C05379=1020.574,11.528,-102.790,166.714,51.533,159.403
C05380=1020.580,11.777,-102.804,166.717,51.528,159.402
C05381=1020.585,12.026,-102.818,166.719,51.522,159.401
C05382=1020.591,12.276,-102.832,166.722,51.517,159.401
C05383=1020.598,12.525,-102.846,166.725,51.512,159.401
C05384=1020.603,12.775,-102.860,166.727,51.506,159.400
C05385=1020.609,13.025,-102.874,166.730,51.501,159.399
C05386=1020.615,13.274,-102.889,166.733,51.496,159.399
C05387=1020.621,13.523,-102.903,166.735,51.491,159.398
C05388=1020.627,13.773,-102.918,166.738,51.485,159.398
C05389=1020.633,14.023,-102.932,166.741,51.480,159.397
C05390=1020.638,14.272,-102.946,166.743,51.475,159.397
C05391=1020.644,14.522,-102.961,166.746,51.469,159.397
C05392=1020.649,14.771,-102.976,166.748,51.465,159.396
C05393=1020.655,15.021,-102.989,166.751,51.459,159.395
C05394=1020.661,15.270,-103.004,166.754,51.453,159.395
C05395=1020.667,15.519,-103.019,166.756,51.448,159.394
C05396=1020.673,15.769,-103.033,166.760,51.443,159.394
C05397=1020.679,16.019,-103.048,166.762,51.438,159.393
C05398=1020.684,16.269,-103.062,166.764,51.432,159.393
C05399=1020.689,16.517,-103.077,166.768,51.427,159.392
C05400=1020.696,16.768,-103.091,166.770,51.422,159.392
C05401=1020.701,17.017,-103.106,166.773,51.417,159.392
C05402=1020.708,17.266,-103.121,166.776,51.411,159.391
C05403=1020.713,17.516,-103.134,166.778,51.406,159.390
C05404=1020.719,17.765,-103.149,166.781,51.401,159.390
C05405=1020.725,18.015,-103.163,166.783,51.396,159.389
C05406=1020.730,18.264,-103.178,166.786,51.390,159.389
C05407=1020.736,18.514,-103.193,166.789,51.385,159.388
C05408=1020.742,18.764,-103.207,166.791,51.380,159.388
C05409=1020.748,19.013,-103.222,166.794,51.374,159.387
C05410=1020.754,19.262,-103.237,166.797,51.369,159.387
C05411=1020.759,19.512,-103.251,166.799,51.364,159.386
C05412=1020.765,19.762,-103.266,166.802,51.359,159.386
C05413=1020.771,20.011,-103.281,166.804,51.354,159.385
C05414=1020.776,20.260,-103.295,166.807,51.348,159.385
C05415=1020.782,20.510,-103.310,166.809,51.343,159.384
C05416=1020.788,20.759,-103.325,166.813,51.338,159.384
C05417=1020.794,21.009,-103.340,166.816,51.333,159.383
C05418=1020.799,21.259,-103.354,166.817,51.327,159.383
C05419=1020.805,21.508,-103.369,166.821,51.322,159.382
C05420=1020.811,21.757,-103.384,166.823,51.317,159.382
C05421=1020.817,22.006,-103.398,166.826,51.312,159.381
C05422=1020.823,22.256,-103.414,166.829,51.306,159.381
C05423=1020.828,22.506,-103.428,166.831,51.301,159.380
C05424=1020.834,22.756,-103.443,166.834,51.296,159.380
C05425=1020.840,23.005,-103.458,166.836,51.291,159.379
C05426=1020.846,23.255,-103.473,166.839,51.285,159.379
C05427=1020.852,23.503,-103.487,166.842,51.280,159.378
C05428=1020.857,23.754,-103.502,166.844,51.275,159.378
C05429=1020.863,24.003,-103.517,166.847,51.269,159.377
C05430=1020.869,24.253,-103.532,166.849,51.265,159.376
C05431=1020.875,24.502,-103.546,166.852,51.259,159.376
C05432=1020.881,24.752,-103.562,166.855,51.253,159.375
C05433=1020.886,25.001,-103.576,166.857,51.249,159.375
C05434=1020.893,25.250,-103.591,166.861,51.243,159.375
C05435=1020.898,25.500,-103.606,166.863,51.237,159.374
C05436=1020.904,25.750,-103.621,166.865,51.233,159.373
C05437=1020.910,25.999,-103.635,166.869,51.227,159.373
C05438=1020.915,26.249,-103.651,166.870,51.222,159.372
C05439=1020.921,26.498,-103.665,166.874,51.217,159.372
C05440=1020.928,26.782,-103.683,166.876,51.211,159.371
C05441=1020.934,27.066,-103.700,166.879,51.205,159.371
C05442=1020.941,27.350,-103.717,166.883,51.199,159.370
C05443=1020.948,27.634,-103.734,166.886,51.193,159.369
C05444=1020.953,27.883,-103.748,166.889,51.187,159.369
C05445=1020.959,28.133,-103.764,166.891,51.182,159.368
C05446=1020.965,28.382,-103.779,166.894,51.177,159.368
C05447=1020.971,28.632,-103.794,166.896,51.172,159.367
C05448=1020.976,28.881,-103.809,166.899,51.166,159.367
C05449=1020.982,29.131,-103.824,166.901,51.161,159.366
C05450=1020.988,29.380,-103.839,166.904,51.156,159.366
C05451=1020.994,29.629,-103.855,166.906,51.151,159.365
C05452=1020.999,29.879,-103.871,166.909,51.145,159.365
C05453=1021.005,30.128,-103.885,166.912,51.140,159.364
C05454=1021.011,30.378,-103.901,166.914,51.135,159.364
C05455=1021.017,30.627,-103.915,166.917,51.129,159.363
C05456=1021.022,30.877,-103.931,166.919,51.125,159.363
C05457=1021.028,31.126,-103.945,166.923,51.119,159.362
C05458=1021.034,31.376,-103.961,166.924,51.114,159.361
C05459=1021.040,31.626,-103.976,166.928,51.109,159.361
C05460=1021.045,31.875,-103.991,166.931,51.103,159.361
C05461=1021.051,32.124,-104.007,166.933,51.098,159.360
C05462=1021.057,32.373,-104.022,166.936,51.093,159.359
C05463=1021.062,32.623,-104.038,166.938,51.088,159.359
C05464=1021.069,32.873,-104.052,166.941,51.082,159.358
C05465=1021.074,33.122,-104.068,166.944,51.077,159.358
C05466=1021.080,33.372,-104.083,166.946,51.072,159.357
C05467=1021.086,33.621,-104.099,166.949,51.066,159.357
C05468=1021.092,33.870,-104.113,166.951,51.061,159.356
C05469=1021.098,34.120,-104.129,166.954,51.056,159.356
C05470=1021.103,34.370,-104.145,166.957,51.050,159.355
C05471=1021.109,34.619,-104.159,166.959,51.045,159.355
C05472=1021.115,34.868,-104.175,166.962,51.040,159.354
C05473=1021.121,35.117,-104.190,166.964,51.035,159.353
C05474=1021.126,35.367,-104.205,166.967,51.030,159.353
C05475=1021.133,35.617,-104.220,166.970,51.024,159.352
C05476=1021.138,35.866,-104.236,166.972,51.019,159.352
C05477=1021.144,36.116,-104.252,166.975,51.013,159.351
C05478=1021.150,36.365,-104.267,166.977,51.008,159.351
C05479=1021.156,36.615,-104.282,166.980,51.002,159.350
C05480=1021.162,36.864,-104.297,166.983,50.997,159.350
C05481=1021.168,37.113,-104.313,166.985,50.992,159.349
C05482=1021.173,37.363,-104.329,166.988,50.986,159.348
C05483=1021.178,37.613,-104.344,166.990,50.982,159.348
C05484=1021.184,37.862,-104.360,166.994,50.976,159.347
C05485=1021.191,38.112,-104.375,166.996,50.972,159.347
C05486=1021.196,38.360,-104.391,166.999,50.966,159.346
C05487=1021.202,38.610,-104.407,167.001,50.961,159.346
C05488=1021.207,38.860,-104.422,167.004,50.956,159.345
C05489=1021.213,39.110,-104.438,167.007,50.950,159.345
C05490=1021.218,39.359,-104.453,167.009,50.945,159.344
C05491=1021.225,39.608,-104.469,167.012,50.940,159.344
C05492=1021.231,39.858,-104.485,167.014,50.934,159.343
C05493=1021.236,40.107,-104.501,167.017,50.929,159.343
C05494=1021.242,40.357,-104.516,167.019,50.924,159.342
C05495=1021.247,40.606,-104.532,167.022,50.918,159.341
C05496=1021.254,40.856,-104.547,167.024,50.914,159.341
C05497=1021.259,41.105,-104.562,167.027,50.908,159.340
C05498=1021.265,41.354,-104.579,167.030,50.903,159.340
C05499=1021.271,41.604,-104.594,167.033,50.898,159.339
C05500=1021.276,41.853,-104.611,167.035,50.892,159.339
C05501=1021.282,42.102,-104.625,167.038,50.887,159.338
C05502=1021.288,42.352,-104.641,167.040,50.881,159.338
C05503=1021.294,42.602,-104.657,167.043,50.876,159.337
C05504=1021.300,42.885,-104.675,167.047,50.870,159.337
C05505=1021.306,43.169,-104.694,167.049,50.864,159.336
C05506=1021.313,43.453,-104.711,167.052,50.859,159.335
C05507=1021.319,43.737,-104.730,167.055,50.853,159.335
C05508=1021.325,43.987,-104.746,167.057,50.848,159.334
C05509=1021.330,44.235,-104.762,167.060,50.843,159.334
C05510=1021.336,44.485,-104.778,167.062,50.837,159.333
C05511=1021.342,44.735,-104.793,167.065,50.832,159.333
C05512=1021.347,44.984,-104.810,167.068,50.827,159.332
C05513=1021.353,45.234,-104.826,167.071,50.822,159.332
C05514=1021.358,45.483,-104.842,167.073,50.817,159.331
C05515=1021.364,45.732,-104.858,167.076,50.812,159.330
C05516=1021.370,45.982,-104.874,167.078,50.807,159.330
C05517=1021.376,46.232,-104.890,167.081,50.801,159.329
C05518=1021.382,46.481,-104.906,167.083,50.796,159.329
C05519=1021.387,46.730,-104.922,167.086,50.791,159.328
C05520=1021.393,46.979,-104.938,167.088,50.785,159.328
C05521=1021.399,47.229,-104.954,167.091,50.780,159.327
C05522=1021.404,47.479,-104.970,167.094,50.775,159.327
C05523=1021.410,47.728,-104.987,167.096,50.770,159.326
C05524=1021.415,47.977,-105.003,167.099,50.765,159.325
C05525=1021.421,48.227,-105.018,167.102,50.760,159.325
C05526=1021.427,48.476,-105.034,167.104,50.754,159.324
C05527=1021.433,48.725,-105.051,167.107,50.749,159.324
C05528=1021.439,48.975,-105.067,167.110,50.744,159.323
C05529=1021.444,49.225,-105.082,167.112,50.738,159.323
C05530=1021.450,49.473,-105.098,167.115,50.733,159.322
C05531=1021.455,49.723,-105.115,167.117,50.728,159.322
C05532=1021.461,49.972,-105.131,167.120,50.723,159.321
C05533=1021.467,50.222,-105.148,167.122,50.718,159.321
C05534=1021.472,50.472,-105.163,167.125,50.712,159.320
C05535=1021.478,50.721,-105.179,167.127,50.707,159.319
C05536=1021.484,50.970,-105.196,167.131,50.702,159.319
C05537=1021.490,51.220,-105.212,167.132,50.697,159.318
C05538=1021.496,51.468,-105.228,167.136,50.691,159.318
C05539=1021.502,51.718,-105.244,167.139,50.686,159.317
C05540=1021.506,51.968,-105.260,167.141,50.681,159.317
C05541=1021.512,52.217,-105.277,167.144,50.675,159.316
C05542=1021.518,52.467,-105.293,167.146,50.670,159.315
C05543=1021.524,52.716,-105.309,167.149,50.665,159.315
C05544=1021.530,52.965,-105.325,167.151,50.660,159.314
C05545=1021.536,53.215,-105.342,167.154,50.654,159.314
C05546=1021.542,53.464,-105.358,167.156,50.649,159.313
C05547=1021.548,53.714,-105.373,167.159,50.644,159.313
C05548=1021.553,53.964,-105.390,167.162,50.638,159.312
C05549=1021.559,54.213,-105.406,167.164,50.633,159.312
C05550=1021.564,54.462,-105.422,167.167,50.627,159.311
C05551=1021.570,54.711,-105.439,167.169,50.623,159.310
C05552=1021.576,54.960,-105.455,167.172,50.617,159.310
C05553=1021.582,55.210,-105.471,167.174,50.612,159.309
C05554=1021.588,55.459,-105.487,167.177,50.606,159.309
C05555=1021.593,55.709,-105.504,167.180,50.601,159.308
C05556=1021.599,55.958,-105.521,167.182,50.596,159.307
C05557=1021.605,56.207,-105.537,167.185,50.590,159.307
C05558=1021.611,56.457,-105.553,167.187,50.585,159.306
C05559=1021.617,56.706,-105.569,167.191,50.580,159.306
C05560=1021.623,56.955,-105.586,167.193,50.574,159.305
C05561=1021.629,57.205,-105.602,167.196,50.569,159.305
C05562=1021.635,57.454,-105.618,167.198,50.563,159.304
C05563=1021.640,57.704,-105.635,167.200,50.558,159.303
C05564=1021.646,57.953,-105.651,167.204,50.553,159.303
C05565=1021.652,58.202,-105.667,167.206,50.547,159.302
C05566=1021.658,58.452,-105.684,167.209,50.542,159.302
C05567=1021.664,58.701,-105.700,167.212,50.536,159.301
C05568=1021.671,58.985,-105.719,167.214,50.531,159.300
C05569=1021.677,59.270,-105.737,167.217,50.525,159.300
C05570=1021.684,59.552,-105.756,167.221,50.518,159.299
C05571=1021.691,59.836,-105.774,167.224,50.512,159.299
C05572=1021.696,60.086,-105.790,167.225,50.507,159.298
C05573=1021.702,60.335,-105.807,167.229,50.502,159.297
C05574=1021.708,60.584,-105.823,167.232,50.496,159.297
C05575=1021.714,60.834,-105.840,167.233,50.490,159.296
C05576=1021.720,61.083,-105.856,167.237,50.485,159.296
C05577=1021.725,61.333,-105.872,167.240,50.479,159.295
C05578=1021.732,61.583,-105.889,167.241,50.474,159.294
C05579=1021.738,61.831,-105.906,167.245,50.469,159.294
C05580=1021.744,62.081,-105.922,167.248,50.463,159.293
C05581=1021.749,62.330,-105.939,167.250,50.458,159.293
C05582=1021.755,62.580,-105.955,167.253,50.453,159.292
C05583=1021.761,62.829,-105.972,167.254,50.447,159.291
C05584=1021.767,63.078,-105.988,167.258,50.442,159.291
C05585=1021.773,63.328,-106.005,167.261,50.436,159.290
C05586=1021.779,63.577,-106.022,167.263,50.431,159.290
C05587=1021.785,63.826,-106.038,167.266,50.426,159.289
C05588=1021.793,64.185,-106.062,167.269,50.418,159.288
C05589=1021.801,64.542,-106.087,167.273,50.410,159.287
C05590=1021.809,64.899,-106.110,167.277,50.403,159.287
C05591=1021.817,65.257,-106.134,167.281,50.396,159.286
C05592=1021.823,65.506,-106.151,167.283,50.390,159.285
C05593=1021.829,65.755,-106.168,167.286,50.385,159.285
C05594=1021.835,66.005,-106.184,167.289,50.379,159.284
C05595=1021.841,66.254,-106.202,167.291,50.375,159.283
C05596=1021.847,66.504,-106.218,167.294,50.369,159.283
C05597=1021.852,66.753,-106.235,167.296,50.364,159.282
C05598=1021.858,67.002,-106.252,167.299,50.358,159.282
C05599=1021.863,67.252,-106.269,167.301,50.353,159.281
C05600=1021.869,67.501,-106.285,167.304,50.348,159.280
C05601=1021.875,67.750,-106.303,167.307,50.343,159.280
C05602=1021.881,68.000,-106.319,167.309,50.337,159.279
C05603=1021.886,68.249,-106.337,167.312,50.331,159.279
C05604=1021.893,68.499,-106.353,167.314,50.327,159.278
C05605=1021.898,68.748,-106.370,167.318,50.322,159.278
C05606=1021.904,68.997,-106.387,167.320,50.316,159.277
C05607=1021.909,69.247,-106.404,167.323,50.311,159.276
C05608=1021.915,69.496,-106.421,167.325,50.306,159.276
C05609=1021.921,69.745,-106.438,167.328,50.300,159.275
C05610=1021.927,69.995,-106.456,167.330,50.295,159.275
C05611=1021.932,70.244,-106.473,167.333,50.290,159.274
C05612=1021.939,70.493,-106.489,167.336,50.284,159.274
C05613=1021.944,70.743,-106.506,167.338,50.279,159.273
C05614=1021.949,70.992,-106.524,167.341,50.274,159.272
C05615=1021.955,71.241,-106.540,167.343,50.269,159.272
C05616=1021.961,71.491,-106.558,167.346,50.263,159.271
C05617=1021.967,71.741,-106.575,167.349,50.258,159.271
C05618=1021.973,71.989,-106.592,167.351,50.253,159.270
C05619=1021.978,72.238,-106.609,167.354,50.248,159.269
C05620=1021.984,72.488,-106.626,167.357,50.242,159.269
C05621=1021.989,72.737,-106.644,167.359,50.237,159.268
C05622=1021.996,72.987,-106.661,167.362,50.232,159.268
C05623=1022.001,73.236,-106.678,167.365,50.227,159.267
C05624=1022.006,73.486,-106.695,167.367,50.221,159.266
C05625=1022.013,73.735,-106.712,167.370,50.216,159.266
C05626=1022.019,73.984,-106.730,167.372,50.211,159.265
C05627=1022.024,74.234,-106.747,167.375,50.205,159.265
C05628=1022.029,74.446,-106.761,167.378,50.201,159.264
C05629=1022.034,74.658,-106.776,167.380,50.196,159.264
C05630=1022.039,74.871,-106.790,167.382,50.191,159.263
C05631=1022.044,75.083,-106.805,167.384,50.188,159.263
C05632=1022.049,75.295,-106.820,167.386,50.183,159.262
C05633=1022.054,75.508,-106.835,167.388,50.178,159.262
C05634=1022.058,75.720,-106.849,167.390,50.173,159.261
C05635=1022.063,75.933,-106.864,167.393,50.169,159.261
C05636=1022.069,76.182,-106.882,167.396,50.163,159.260
C05637=1022.075,76.431,-106.898,167.398,50.159,159.260
C05638=1022.081,76.681,-106.916,167.401,50.153,159.259
C05639=1022.087,76.930,-106.933,167.403,50.148,159.258
C05640=1022.092,77.179,-106.951,167.406,50.142,159.258
C05641=1022.097,77.429,-106.968,167.409,50.138,159.257
C05642=1022.103,77.679,-106.986,167.411,50.132,159.257
C05643=1022.109,77.928,-107.003,167.414,50.127,159.256
C05644=1022.114,78.177,-107.021,167.417,50.122,159.255
C05645=1022.120,78.426,-107.038,167.420,50.116,159.255
C05646=1022.126,78.676,-107.056,167.422,50.111,159.254
C05647=1022.131,78.925,-107.073,167.425,50.106,159.254
C05648=1022.137,79.174,-107.091,167.427,50.101,159.253
C05649=1022.143,79.424,-107.109,167.430,50.096,159.253
C05650=1022.149,79.673,-107.126,167.433,50.091,159.252
C05651=1022.155,79.922,-107.143,167.435,50.085,159.252
C05652=1022.160,80.171,-107.160,167.438,50.080,159.251
C05653=1022.166,80.421,-107.178,167.441,50.075,159.250
C05654=1022.172,80.670,-107.196,167.443,50.070,159.250
C05655=1022.177,80.919,-107.213,167.446,50.064,159.249
C05656=1022.183,81.169,-107.231,167.448,50.059,159.249
C05657=1022.189,81.418,-107.249,167.451,50.054,159.248
C05658=1022.194,81.667,-107.266,167.453,50.049,159.247
C05659=1022.200,81.916,-107.284,167.456,50.043,159.247
C05660=1022.206,82.166,-107.302,167.459,50.038,159.246
C05661=1022.211,82.415,-107.319,167.461,50.033,159.246
C05662=1022.217,82.664,-107.337,167.465,50.028,159.245
C05663=1022.223,82.914,-107.354,167.467,50.022,159.244
C05664=1022.228,83.163,-107.372,167.470,50.017,159.244
C05665=1022.234,83.412,-107.389,167.472,50.012,159.243
C05666=1022.240,83.662,-107.407,167.475,50.007,159.243
C05667=1022.245,83.911,-107.425,167.478,50.001,159.242
C05668=1022.252,84.161,-107.443,167.480,49.996,159.241
C05669=1022.257,84.410,-107.460,167.483,49.991,159.241
C05670=1022.263,84.659,-107.478,167.485,49.985,159.240
C05671=1022.269,84.909,-107.496,167.488,49.980,159.240
C05672=1022.274,85.158,-107.513,167.490,49.975,159.239
C05673=1022.280,85.407,-107.531,167.494,49.970,159.239
C05674=1022.286,85.656,-107.549,167.497,49.964,159.238
C05675=1022.291,85.906,-107.566,167.499,49.959,159.237
C05676=1022.297,86.155,-107.584,167.502,49.953,159.237
C05677=1022.303,86.404,-107.602,167.504,49.948,159.236
C05678=1022.309,86.653,-107.619,167.507,49.943,159.236
C05679=1022.315,86.903,-107.637,167.510,49.937,159.235
C05680=1022.320,87.152,-107.655,167.512,49.933,159.234
C05681=1022.326,87.402,-107.673,167.515,49.927,159.234
C05682=1022.332,87.651,-107.690,167.517,49.921,159.233
C05683=1022.338,87.899,-107.709,167.520,49.916,159.233
C05684=1022.344,88.149,-107.727,167.523,49.911,159.232
C05685=1022.349,88.398,-107.744,167.526,49.906,159.231
C05686=1022.355,88.648,-107.762,167.529,49.900,159.231
C05687=1022.361,88.897,-107.780,167.530,49.895,159.230
C05688=1022.367,89.147,-107.798,167.534,49.890,159.230
C05689=1022.372,89.396,-107.816,167.537,49.884,159.229
C05690=1022.378,89.646,-107.834,167.539,49.879,159.228
C05691=1022.383,89.895,-107.851,167.542,49.874,159.228
C05692=1022.389,90.143,-107.870,167.544,49.869,159.227
C05693=1022.395,90.393,-107.888,167.547,49.863,159.227
C05694=1022.400,90.642,-107.906,167.549,49.859,159.226
C05695=1022.406,90.892,-107.924,167.552,49.853,159.225
C05696=1022.413,91.175,-107.944,167.555,49.847,159.225
C05697=1022.419,91.459,-107.965,167.558,49.841,159.224
C05698=1022.425,91.742,-107.986,167.561,49.836,159.224
C05699=1022.432,92.026,-108.007,167.565,49.829,159.223
C05700=1022.437,92.275,-108.025,167.567,49.824,159.222
C05701=1022.443,92.525,-108.043,167.570,49.819,159.222
C05702=1022.448,92.774,-108.061,167.572,49.814,159.221
C05703=1022.455,93.023,-108.079,167.575,49.808,159.221
C05704=1022.460,93.272,-108.097,167.578,49.804,159.220
C05705=1022.466,93.522,-108.115,167.581,49.798,159.219
C05706=1022.471,93.771,-108.134,167.584,49.793,159.219
C05707=1022.477,94.020,-108.151,167.586,49.787,159.218
C05708=1022.483,94.270,-108.169,167.589,49.782,159.218
C05709=1022.488,94.518,-108.188,167.591,49.777,159.217
C05710=1022.494,94.768,-108.206,167.594,49.772,159.217
C05711=1022.500,95.016,-108.224,167.596,49.767,159.216
C05712=1022.505,95.267,-108.243,167.600,49.762,159.215
C05713=1022.511,95.516,-108.261,167.603,49.756,159.215
C05714=1022.517,95.765,-108.279,167.605,49.751,159.214
C05715=1022.523,96.015,-108.298,167.608,49.746,159.214
C05716=1022.528,96.264,-108.315,167.610,49.740,159.213
C05717=1022.535,96.513,-108.334,167.613,49.735,159.212
C05718=1022.539,96.762,-108.352,167.616,49.729,159.212
C05719=1022.546,97.011,-108.371,167.618,49.725,159.211
C05720=1022.551,97.260,-108.388,167.621,49.719,159.211
C05721=1022.557,97.510,-108.408,167.624,49.714,159.210
C05722=1022.563,97.759,-108.425,167.627,49.709,159.209
C05723=1022.569,98.009,-108.443,167.630,49.703,159.209
C05724=1022.574,98.258,-108.462,167.632,49.698,159.208
C05725=1022.580,98.507,-108.480,167.635,49.693,159.207
C05726=1022.586,98.756,-108.498,167.638,49.688,159.207
C05727=1022.591,99.006,-108.517,167.640,49.682,159.206
C05728=1022.597,99.255,-108.535,167.643,49.677,159.206
C05729=1022.603,99.504,-108.553,167.645,49.672,159.205
C05730=1022.609,99.753,-108.572,167.648,49.666,159.204
C05731=1022.614,100.003,-108.591,167.652,49.661,159.204
C05732=1022.620,100.252,-108.609,167.654,49.657,159.203
C05733=1022.626,100.501,-108.628,167.657,49.651,159.203
C05734=1022.631,100.750,-108.646,167.659,49.646,159.202
C05735=1022.637,101.000,-108.665,167.662,49.640,159.202
C05736=1022.642,101.249,-108.683,167.665,49.636,159.201
C05737=1022.648,101.498,-108.702,167.668,49.630,159.200
C05738=1022.654,101.747,-108.721,167.670,49.625,159.200
C05739=1022.659,101.997,-108.739,167.673,49.620,159.199
C05740=1022.665,102.246,-108.758,167.676,49.615,159.199
C05741=1022.670,102.495,-108.777,167.678,49.609,159.198
C05742=1022.676,102.744,-108.795,167.681,49.604,159.198
C05743=1022.682,102.994,-108.814,167.683,49.599,159.197
C05744=1022.687,103.243,-108.833,167.687,49.594,159.196
C05745=1022.693,103.492,-108.851,167.690,49.588,159.196
C05746=1022.699,103.742,-108.870,167.692,49.584,159.195
C05747=1022.704,103.990,-108.888,167.695,49.578,159.195
C05748=1022.710,104.240,-108.907,167.697,49.573,159.194
C05749=1022.715,104.489,-108.926,167.700,49.568,159.193
C05750=1022.721,104.738,-108.944,167.703,49.563,159.193
C05751=1022.727,104.988,-108.964,167.706,49.557,159.192
C05752=1022.732,105.237,-108.982,167.709,49.552,159.192
C05753=1022.738,105.486,-109.000,167.711,49.547,159.191
C05754=1022.744,105.735,-109.020,167.714,49.542,159.191
C05755=1022.750,105.984,-109.038,167.717,49.536,159.190
C05756=1022.755,106.233,-109.057,167.720,49.532,159.189
C05757=1022.761,106.483,-109.076,167.723,49.526,159.189
C05758=1022.767,106.732,-109.094,167.725,49.521,159.188
C05759=1022.772,106.981,-109.113,167.728,49.516,159.188
C05760=1022.779,107.265,-109.134,167.731,49.510,159.187
C05761=1022.785,107.549,-109.155,167.735,49.504,159.186
C05762=1022.792,107.832,-109.177,167.737,49.498,159.186
C05763=1022.799,108.116,-109.199,167.740,49.492,159.185
C05764=1022.804,108.365,-109.217,167.743,49.486,159.184
C05765=1022.810,108.614,-109.236,167.746,49.482,159.184
C05766=1022.815,108.864,-109.255,167.749,49.476,159.183
C05767=1022.821,109.113,-109.273,167.752,49.471,159.183
C05768=1022.827,109.362,-109.292,167.754,49.466,159.182
C05769=1022.833,109.612,-109.312,167.757,49.460,159.181
C05770=1022.839,109.861,-109.330,167.760,49.455,159.181
C05771=1022.844,110.109,-109.349,167.762,49.450,159.180
C05772=1022.850,110.359,-109.368,167.766,49.445,159.180
C05773=1022.856,110.608,-109.388,167.769,49.439,159.179
C05774=1022.861,110.858,-109.407,167.771,49.434,159.178
C05775=1022.867,111.106,-109.425,167.774,49.429,159.178
C05776=1022.873,111.356,-109.444,167.776,49.424,159.177
C05777=1022.878,111.605,-109.464,167.779,49.419,159.177
C05778=1022.884,111.854,-109.483,167.783,49.414,159.176
C05779=1022.889,112.103,-109.502,167.785,49.408,159.175
C05780=1022.895,112.353,-109.521,167.788,49.403,159.175
C05781=1022.901,112.602,-109.540,167.791,49.398,159.174
C05782=1022.906,112.851,-109.559,167.793,49.393,159.174
C05783=1022.911,113.100,-109.578,167.797,49.388,159.173
C05784=1022.917,113.350,-109.598,167.799,49.383,159.173
C05785=1022.923,113.599,-109.617,167.802,49.378,159.172
C05786=1022.928,113.848,-109.636,167.804,49.373,159.172
C05787=1022.933,114.097,-109.655,167.807,49.367,159.171
C05788=1022.939,114.346,-109.675,167.810,49.363,159.170
C05789=1022.945,114.595,-109.694,167.813,49.358,159.170
C05790=1022.951,114.845,-109.713,167.816,49.352,159.169
C05791=1022.956,115.094,-109.732,167.818,49.348,159.169
C05792=1022.961,115.343,-109.752,167.822,49.342,159.168
C05793=1022.967,115.593,-109.771,167.824,49.337,159.168
C05794=1022.973,115.842,-109.791,167.827,49.332,159.167
C05795=1022.978,116.091,-109.811,167.830,49.327,159.166
C05796=1022.983,116.340,-109.829,167.833,49.322,159.166
C05797=1022.989,116.589,-109.849,167.836,49.317,159.165
C05798=1022.995,116.838,-109.869,167.838,49.312,159.165
C05799=1023.001,117.087,-109.888,167.841,49.307,159.164
C05800=1023.006,117.337,-109.907,167.844,49.301,159.164
C05801=1023.011,117.586,-109.927,167.847,49.297,159.163
C05802=1023.017,117.835,-109.947,167.850,49.292,159.163
C05803=1023.022,118.084,-109.966,167.852,49.286,159.162
C05804=1023.028,118.334,-109.985,167.855,49.281,159.161
C05805=1023.034,118.583,-110.004,167.858,49.276,159.161
C05806=1023.039,118.831,-110.024,167.861,49.271,159.160
C05807=1023.045,119.081,-110.043,167.864,49.265,159.160
C05808=1023.051,119.330,-110.062,167.867,49.260,159.159
C05809=1023.056,119.579,-110.082,167.869,49.256,159.159
C05810=1023.062,119.829,-110.102,167.872,49.250,159.158
C05811=1023.067,120.078,-110.121,167.876,49.245,159.157
C05812=1023.073,120.327,-110.141,167.878,49.240,159.157
C05813=1023.078,120.576,-110.160,167.881,49.235,159.156
C05814=1023.084,120.825,-110.179,167.883,49.230,159.156
C05815=1023.090,121.074,-110.199,167.887,49.225,159.155
C05816=1023.096,121.323,-110.219,167.890,49.219,159.154
C05817=1023.101,121.573,-110.238,167.892,49.215,159.154
C05818=1023.107,121.822,-110.258,167.895,49.210,159.153
C05819=1023.112,122.071,-110.278,167.898,49.204,159.153
C05820=1023.118,122.321,-110.297,167.901,49.199,159.152
C05821=1023.124,122.569,-110.317,167.904,49.194,159.152
C05822=1023.130,122.819,-110.336,167.907,49.189,159.151
C05823=1023.135,123.068,-110.355,167.910,49.183,159.150
C05824=1023.141,123.351,-110.377,167.913,49.178,159.150
C05825=1023.148,123.635,-110.400,167.916,49.172,159.149
C05826=1023.154,123.919,-110.422,167.920,49.165,159.148
C05827=1023.161,124.202,-110.444,167.923,49.160,159.148
C05828=1023.167,124.451,-110.464,167.926,49.155,159.147
C05829=1023.172,124.701,-110.484,167.928,49.150,159.147
C05830=1023.178,124.950,-110.504,167.932,49.145,159.146
C05831=1023.184,125.199,-110.523,167.935,49.139,159.146
C05832=1023.190,125.448,-110.543,167.937,49.134,159.145
C05833=1023.195,125.697,-110.563,167.940,49.129,159.144
C05834=1023.201,125.946,-110.582,167.943,49.124,159.144
C05835=1023.207,126.196,-110.602,167.947,49.118,159.143
C05836=1023.212,126.445,-110.622,167.949,49.114,159.143
C05837=1023.218,126.694,-110.642,167.952,49.108,159.142
C05838=1023.224,126.943,-110.661,167.955,49.103,159.142
C05839=1023.230,127.192,-110.681,167.957,49.098,159.141
C05840=1023.236,127.441,-110.701,167.961,49.093,159.140
C05841=1023.241,127.691,-110.720,167.964,49.087,159.140
C05842=1023.247,127.939,-110.740,167.967,49.082,159.139
C05843=1023.252,128.189,-110.760,167.969,49.077,159.139
C05844=1023.258,128.438,-110.780,167.973,49.072,159.138
C05845=1023.264,128.687,-110.799,167.976,49.067,159.137
C05846=1023.270,128.936,-110.819,167.979,49.061,159.137
C05847=1023.276,129.186,-110.838,167.981,49.056,159.136
C05848=1023.282,129.434,-110.858,167.984,49.051,159.136
C05849=1023.288,129.683,-110.878,167.987,49.046,159.135
C05850=1023.292,129.933,-110.898,167.990,49.040,159.134
C05851=1023.298,130.182,-110.918,167.993,49.036,159.134
C05852=1023.304,130.431,-110.938,167.996,49.031,159.133
C05853=1023.309,130.680,-110.958,167.999,49.025,159.133
C05854=1023.315,130.929,-110.978,168.003,49.020,159.132
C05855=1023.321,131.178,-110.998,168.005,49.015,159.132
C05856=1023.327,131.427,-111.018,168.008,49.010,159.131
C05857=1023.332,131.677,-111.038,168.011,49.005,159.131
C05858=1023.338,131.926,-111.058,168.013,49.000,159.130
C05859=1023.343,132.175,-111.078,168.017,48.995,159.129
C05860=1023.349,132.424,-111.098,168.020,48.990,159.129
C05861=1023.354,132.673,-111.119,168.022,48.985,159.128
C05862=1023.360,132.922,-111.138,168.026,48.980,159.128
C05863=1023.365,133.171,-111.159,168.029,48.974,159.127
C05864=1023.372,133.421,-111.179,168.032,48.969,159.127
C05865=1023.377,133.670,-111.200,168.034,48.965,159.126
C05866=1023.383,133.919,-111.220,168.038,48.959,159.125
C05867=1023.388,134.168,-111.240,168.041,48.954,159.125
C05868=1023.394,134.417,-111.259,168.043,48.950,159.124
C05869=1023.399,134.666,-111.280,168.046,48.944,159.124
C05870=1023.405,134.915,-111.300,168.050,48.939,159.123
C05871=1023.410,135.164,-111.320,168.053,48.934,159.123
C05872=1023.416,135.413,-111.340,168.055,48.929,159.122
C05873=1023.422,135.662,-111.361,168.059,48.924,159.122
C05874=1023.428,135.911,-111.381,168.062,48.919,159.121
C05875=1023.433,136.161,-111.402,168.065,48.914,159.121
C05876=1023.439,136.410,-111.421,168.067,48.908,159.120
C05877=1023.444,136.659,-111.442,168.071,48.903,159.119
C05878=1023.450,136.908,-111.462,168.074,48.899,159.119
C05879=1023.456,137.157,-111.482,168.077,48.893,159.118
C05880=1023.461,137.407,-111.503,168.079,48.888,159.118
C05881=1023.467,137.655,-111.523,168.083,48.884,159.117
C05882=1023.473,137.905,-111.544,168.086,48.878,159.117
C05883=1023.479,138.154,-111.564,168.089,48.873,159.116
C05884=1023.484,138.403,-111.584,168.092,48.868,159.116
C05885=1023.489,138.652,-111.605,168.095,48.863,159.115
C05886=1023.495,138.901,-111.625,168.098,48.858,159.114
C05887=1023.500,139.150,-111.645,168.101,48.853,159.114
C05888=1023.507,139.434,-111.669,168.105,48.848,159.113
C05889=1023.513,139.718,-111.693,168.108,48.842,159.113
C05890=1023.520,140.001,-111.716,168.112,48.836,159.112
C05891=1023.526,140.284,-111.739,168.115,48.831,159.111
C05892=1023.532,140.533,-111.760,168.118,48.825,159.111
C05893=1023.537,140.782,-111.781,168.121,48.820,159.110
C05894=1023.543,141.031,-111.801,168.124,48.816,159.110
C05895=1023.549,141.281,-111.821,168.127,48.810,159.109
C05896=1023.554,141.530,-111.842,168.130,48.805,159.109
C05897=1023.559,141.779,-111.863,168.134,48.800,159.108
C05898=1023.565,142.027,-111.883,168.136,48.796,159.108
C05899=1023.571,142.276,-111.904,168.139,48.790,159.107
C05900=1023.577,142.526,-111.925,168.142,48.785,159.107
C05901=1023.582,142.775,-111.945,168.146,48.780,159.106
C05902=1023.588,143.024,-111.965,168.148,48.775,159.105
C05903=1023.593,143.273,-111.987,168.151,48.770,159.105
C05904=1023.599,143.522,-112.007,168.155,48.765,159.104
C05905=1023.605,143.772,-112.028,168.158,48.760,159.104
C05906=1023.611,144.020,-112.048,168.161,48.755,159.103
C05907=1023.616,144.269,-112.069,168.164,48.750,159.103
C05908=1023.622,144.519,-112.090,168.167,48.745,159.102
C05909=1023.627,144.768,-112.111,168.170,48.740,159.102
C05910=1023.632,145.017,-112.131,168.174,48.735,159.101
C05911=1023.639,145.265,-112.152,168.177,48.730,159.100
C05912=1023.645,145.515,-112.173,168.179,48.725,159.100
C05913=1023.650,145.764,-112.193,168.182,48.720,159.099
C05914=1023.655,146.013,-112.214,168.185,48.715,159.099
C05915=1023.661,146.262,-112.236,168.189,48.710,159.098
C05916=1023.667,146.512,-112.256,168.192,48.705,159.098
C05917=1023.672,146.760,-112.277,168.195,48.700,159.097
C05918=1023.678,147.009,-112.297,168.198,48.695,159.097
C05919=1023.684,147.259,-112.318,168.201,48.690,159.096
C05920=1023.689,147.507,-112.340,168.205,48.685,159.096
C05921=1023.695,147.756,-112.360,168.208,48.680,159.095
C05922=1023.701,148.006,-112.382,168.210,48.676,159.095
C05923=1023.706,148.255,-112.402,168.214,48.670,159.094
C05924=1023.712,148.503,-112.424,168.217,48.665,159.094
C05925=1023.717,148.752,-112.444,168.220,48.660,159.093
C05926=1023.723,149.002,-112.465,168.224,48.655,159.093
C05927=1023.728,149.251,-112.486,168.226,48.650,159.092
C05928=1023.734,149.500,-112.507,168.229,48.645,159.091
C05929=1023.740,149.749,-112.528,168.233,48.641,159.091
C05930=1023.745,149.998,-112.549,168.236,48.636,159.090
C05931=1023.751,150.247,-112.570,168.240,48.631,159.090
C05932=1023.756,150.496,-112.593,168.242,48.626,159.089
C05933=1023.761,150.745,-112.613,168.245,48.621,159.089
C05934=1023.767,150.994,-112.634,168.249,48.616,159.088
C05935=1023.773,151.244,-112.655,168.252,48.611,159.088
C05936=1023.778,151.492,-112.677,168.255,48.606,159.087
C05937=1023.784,151.742,-112.697,168.258,48.601,159.087
C05938=1023.790,151.990,-112.719,168.261,48.596,159.086
C05939=1023.795,152.240,-112.739,168.264,48.591,159.086
C05940=1023.801,152.489,-112.761,168.268,48.586,159.085
C05941=1023.807,152.737,-112.782,168.271,48.581,159.085
C05942=1023.812,152.986,-112.803,168.274,48.576,159.084
C05943=1023.818,153.236,-112.824,168.278,48.571,159.084
C05944=1023.824,153.484,-112.846,168.280,48.567,159.083
C05945=1023.830,153.734,-112.867,168.284,48.562,159.083
C05946=1023.834,153.983,-112.888,168.287,48.557,159.082
C05947=1023.841,154.232,-112.910,168.290,48.551,159.081
C05948=1023.846,154.481,-112.931,168.294,48.547,159.081
C05949=1023.851,154.730,-112.952,168.297,48.542,159.080
C05950=1023.858,154.979,-112.974,168.299,48.537,159.080
C05951=1023.862,155.228,-112.995,168.303,48.532,159.079
C05952=1023.869,155.512,-113.019,168.307,48.527,159.079
C05953=1023.875,155.794,-113.044,168.310,48.521,159.078
C05954=1023.882,156.078,-113.067,168.314,48.515,159.078
C05955=1023.888,156.360,-113.092,168.317,48.510,159.077
C05956=1023.894,156.610,-113.113,168.321,48.505,159.077
C05957=1023.899,156.858,-113.135,168.324,48.500,159.076
C05958=1023.905,157.108,-113.156,168.328,48.495,159.076
C05959=1023.910,157.357,-113.177,168.331,48.490,159.075
C05960=1023.917,157.606,-113.199,168.334,48.486,159.075
C05961=1023.921,157.855,-113.221,168.338,48.480,159.074
C05962=1023.928,158.104,-113.243,168.341,48.475,159.074
C05963=1023.933,158.352,-113.264,168.343,48.471,159.073
C05964=1023.939,158.602,-113.285,168.347,48.466,159.072
C05965=1023.945,158.851,-113.306,168.350,48.461,159.072
C05966=1023.950,159.100,-113.328,168.354,48.456,159.072
C05967=1023.956,159.349,-113.350,168.357,48.451,159.071
C05968=1023.961,159.598,-113.372,168.361,48.447,159.071
C05969=1023.967,159.847,-113.393,168.364,48.442,159.070
C05970=1023.972,160.096,-113.415,168.367,48.437,159.070
C05971=1023.977,160.345,-113.437,168.370,48.432,159.069
C05972=1023.983,160.594,-113.459,168.373,48.428,159.069
C05973=1023.988,160.843,-113.481,168.377,48.423,159.068
C05974=1023.993,161.091,-113.503,168.380,48.418,159.068
C05975=1023.999,161.341,-113.525,168.383,48.413,159.067
C05976=1024.004,161.589,-113.547,168.386,48.409,159.067
C05977=1024.009,161.839,-113.569,168.390,48.404,159.066
C05978=1024.015,162.087,-113.590,168.393,48.400,159.066
C05979=1024.020,162.337,-113.612,168.397,48.395,159.065
C05980=1024.025,162.585,-113.635,168.400,48.390,159.065
C05981=1024.032,162.834,-113.657,168.403,48.385,159.064
C05982=1024.037,163.084,-113.679,168.406,48.381,159.064
C05983=1024.042,163.333,-113.701,168.410,48.376,159.063
C05984=1024.048,163.582,-113.722,168.413,48.371,159.063
C05985=1024.053,163.831,-113.744,168.417,48.366,159.062
C05986=1024.059,164.080,-113.767,168.420,48.361,159.062
C05987=1024.064,164.328,-113.788,168.423,48.357,159.061
C05988=1024.070,164.578,-113.811,168.426,48.352,159.061
C05989=1024.074,164.826,-113.833,168.429,48.347,159.060
C05990=1024.081,165.075,-113.855,168.433,48.342,159.060
C05991=1024.086,165.325,-113.877,168.436,48.338,159.059
C05992=1024.091,165.573,-113.899,168.440,48.333,159.059
C05993=1024.097,165.823,-113.921,168.443,48.329,159.059
C05994=1024.102,166.071,-113.943,168.447,48.324,159.058
C05995=1024.108,166.320,-113.965,168.450,48.319,159.058
C05996=1024.113,166.569,-113.987,168.454,48.314,159.057
C05997=1024.119,166.818,-114.010,168.457,48.309,159.057
C05998=1024.125,167.067,-114.032,168.460,48.305,159.056
C05999=1024.130,167.316,-114.053,168.463,48.300,159.056
C06000=1024.135,167.565,-114.075,168.467,48.295,159.055
C06001=1024.141,167.814,-114.098,168.470,48.290,159.055
C06002=1024.146,168.063,-114.120,168.474,48.286,159.054
C06003=1024.153,168.311,-114.143,168.477,48.281,159.054
C06004=1024.158,168.561,-114.165,168.480,48.276,159.053
C06005=1024.163,168.810,-114.187,168.484,48.271,159.053
C06006=1024.169,169.058,-114.209,168.488,48.267,159.052
C06007=1024.175,169.308,-114.231,168.491,48.262,159.052
C06008=1024.179,169.557,-114.253,168.495,48.258,159.052
C06009=1024.186,169.805,-114.275,168.498,48.253,159.051
C06010=1024.191,170.055,-114.298,168.502,48.248,159.051
C06011=1024.197,170.303,-114.320,168.505,48.243,159.050
C06012=1024.203,170.552,-114.342,168.509,48.238,159.050
C06013=1024.208,170.802,-114.364,168.512,48.234,159.049
C06014=1024.213,171.050,-114.387,168.515,48.229,159.049
C06015=1024.219,171.299,-114.409,168.519,48.224,159.048
C06016=1024.226,171.582,-114.434,168.522,48.219,159.048
C06017=1024.232,171.865,-114.460,168.527,48.213,159.047
C06018=1024.238,172.147,-114.484,168.531,48.208,159.047
C06019=1024.245,172.431,-114.510,168.534,48.203,159.046
C06020=1024.250,172.680,-114.533,168.538,48.198,159.046
C06021=1024.256,172.928,-114.555,168.541,48.193,159.045
C06022=1024.262,173.177,-114.577,168.545,48.189,159.045
C06023=1024.267,173.426,-114.600,168.548,48.184,159.044
C06024=1024.273,173.676,-114.622,168.551,48.179,159.044
C06025=1024.279,173.924,-114.644,168.555,48.174,159.043
C06026=1024.284,174.173,-114.667,168.558,48.169,159.043
C06027=1024.290,174.422,-114.689,168.563,48.164,159.042
C06028=1024.296,174.671,-114.712,168.566,48.160,159.042
C06029=1024.302,174.920,-114.734,168.570,48.155,159.041
C06030=1024.308,175.169,-114.757,168.574,48.151,159.041
C06031=1024.312,175.418,-114.779,168.577,48.146,159.040
C06032=1024.319,175.667,-114.801,168.581,48.141,159.040
C06033=1024.325,175.915,-114.824,168.584,48.136,159.040
C06034=1024.330,176.165,-114.846,168.588,48.132,159.039
C06035=1024.336,176.414,-114.868,168.591,48.127,159.039
C06036=1024.342,176.662,-114.891,168.594,48.122,159.038
C06037=1024.347,176.911,-114.913,168.598,48.117,159.038
C06038=1024.353,177.160,-114.936,168.601,48.112,159.037
C06039=1024.359,177.409,-114.959,168.605,48.108,159.037
C06040=1024.365,177.658,-114.981,168.608,48.103,159.036
C06041=1024.370,177.907,-115.004,168.613,48.098,159.036
C06042=1024.377,178.156,-115.026,168.617,48.094,159.035
C06043=1024.382,178.405,-115.048,168.620,48.089,159.035
C06044=1024.388,178.654,-115.071,168.624,48.084,159.034
C06045=1024.393,178.902,-115.094,168.627,48.079,159.034
C06046=1024.400,179.151,-115.116,168.631,48.075,159.033
C06047=1024.405,179.400,-115.138,168.634,48.070,159.033
C06048=1024.411,179.649,-115.161,168.638,48.065,159.032
C06049=1024.416,179.898,-115.184,168.641,48.060,159.032
C06050=1024.423,180.147,-115.207,168.645,48.055,159.032
C06051=1024.428,180.396,-115.229,168.649,48.051,159.031
C06052=1024.434,180.645,-115.252,168.653,48.046,159.031
C06053=1024.440,180.894,-115.275,168.656,48.042,159.030
C06054=1024.446,181.143,-115.297,168.660,48.037,159.030
C06055=1024.452,181.392,-115.320,168.663,48.032,159.029
C06056=1024.458,181.641,-115.343,168.667,48.027,159.029
C06057=1024.464,181.890,-115.365,168.671,48.022,159.028
C06058=1024.470,182.139,-115.388,168.675,48.018,159.028
C06059=1024.475,182.388,-115.411,168.678,48.013,159.027
C06060=1024.481,182.636,-115.434,168.682,48.009,159.027
C06061=1024.486,182.886,-115.457,168.685,48.004,159.027
C06062=1024.492,183.135,-115.480,168.689,47.999,159.026
C06063=1024.498,183.383,-115.503,168.693,47.995,159.026
C06064=1024.503,183.633,-115.526,168.696,47.990,159.025
C06065=1024.509,183.881,-115.550,168.700,47.986,159.025
C06066=1024.514,184.130,-115.573,168.703,47.982,159.025
C06067=1024.519,184.379,-115.597,168.707,47.977,159.024
C06068=1024.524,184.627,-115.619,168.711,47.973,159.024
C06069=1024.530,184.876,-115.642,168.716,47.968,159.024
C06070=1024.535,185.125,-115.666,168.719,47.964,159.023
C06071=1024.541,185.374,-115.689,168.723,47.959,159.023
C06072=1024.547,185.622,-115.712,168.726,47.955,159.022
C06073=1024.552,185.872,-115.736,168.730,47.950,159.022
C06074=1024.558,186.121,-115.759,168.734,47.946,159.021
C06075=1024.563,186.369,-115.783,168.737,47.941,159.021
C06076=1024.569,186.618,-115.806,168.741,47.937,159.021
C06077=1024.574,186.867,-115.829,168.744,47.932,159.020
C06078=1024.580,187.116,-115.853,168.748,47.928,159.020
C06079=1024.585,187.364,-115.876,168.752,47.923,159.019
C06080=1024.592,187.647,-115.903,168.756,47.918,159.019
C06081=1024.598,187.930,-115.929,168.761,47.913,159.019
C06082=1024.604,188.212,-115.956,168.765,47.908,159.018
C06083=1024.611,188.494,-115.982,168.769,47.903,159.018
C06084=1024.617,188.743,-116.005,168.773,47.899,159.017
C06085=1024.622,188.992,-116.030,168.777,47.894,159.017
C06086=1024.628,189.241,-116.053,168.781,47.890,159.016
C06087=1024.633,189.490,-116.076,168.784,47.885,159.016
C06088=1024.639,189.738,-116.100,168.788,47.881,159.016
C06089=1024.645,189.987,-116.123,168.792,47.876,159.015
C06090=1024.650,190.237,-116.146,168.796,47.872,159.015
C06091=1024.656,190.485,-116.170,168.800,47.867,159.014
C06092=1024.662,190.734,-116.193,168.804,47.863,159.014
C06093=1024.667,190.982,-116.217,168.807,47.858,159.014
C06094=1024.673,191.231,-116.240,168.811,47.854,159.013
C06095=1024.679,191.481,-116.265,168.815,47.849,159.013
C06096=1024.684,191.729,-116.288,168.819,47.845,159.013
C06097=1024.690,191.978,-116.311,168.823,47.841,159.012
C06098=1024.695,192.227,-116.335,168.826,47.836,159.012
C06099=1024.701,192.475,-116.359,168.830,47.832,159.011
C06100=1024.706,192.724,-116.382,168.835,47.827,159.011
C06101=1024.713,192.973,-116.406,168.838,47.823,159.010
C06102=1024.719,193.222,-116.429,168.842,47.818,159.010
C06103=1024.724,193.471,-116.453,168.846,47.814,159.010
C06104=1024.730,193.720,-116.476,168.849,47.809,159.009
C06105=1024.735,193.968,-116.501,168.854,47.805,159.009
C06106=1024.741,194.217,-116.524,168.857,47.800,159.008
C06107=1024.747,194.466,-116.548,168.861,47.796,159.008
C06108=1024.753,194.715,-116.572,168.865,47.792,159.008
C06109=1024.758,194.964,-116.595,168.870,47.787,159.007
C06110=1024.765,195.212,-116.619,168.873,47.783,159.007
C06111=1024.770,195.462,-116.642,168.877,47.778,159.007
C06112=1024.776,195.710,-116.666,168.881,47.774,159.006
C06113=1024.781,195.959,-116.690,168.885,47.769,159.006
C06114=1024.787,196.208,-116.713,168.889,47.765,159.006
C06115=1024.793,196.457,-116.738,168.893,47.760,159.005
C06116=1024.799,196.705,-116.762,168.897,47.756,159.005
C06117=1024.805,196.954,-116.785,168.901,47.751,159.004
C06118=1024.810,197.203,-116.809,168.905,47.747,159.004
C06119=1024.817,197.452,-116.833,168.908,47.743,159.003
C06120=1024.822,197.701,-116.856,168.913,47.738,159.003
C06121=1024.828,197.949,-116.880,168.917,47.733,159.003
C06122=1024.834,198.198,-116.904,168.920,47.729,159.002
C06123=1024.840,198.447,-116.928,168.925,47.725,159.002
C06124=1024.845,198.696,-116.951,168.929,47.720,159.002
C06125=1024.851,198.945,-116.976,168.933,47.716,159.001
C06126=1024.857,199.193,-117.000,168.937,47.711,159.001
C06127=1024.863,199.441,-117.023,168.941,47.707,159.001
C06128=1024.869,199.691,-117.048,168.944,47.703,159.000
C06129=1024.875,199.940,-117.071,168.949,47.698,159.000
C06130=1024.881,200.189,-117.095,168.953,47.694,159.000
C06131=1024.886,200.438,-117.120,168.957,47.690,158.999
C06132=1024.892,200.686,-117.144,168.961,47.685,158.999
C06133=1024.898,200.935,-117.168,168.965,47.681,158.998
C06134=1024.904,201.184,-117.192,168.969,47.677,158.998
C06135=1024.909,201.432,-117.216,168.973,47.672,158.998
C06136=1024.915,201.682,-117.241,168.977,47.668,158.997
C06137=1024.920,201.930,-117.265,168.981,47.664,158.997
C06138=1024.926,202.178,-117.289,168.985,47.660,158.997
C06139=1024.932,202.428,-117.314,168.990,47.656,158.996
C06140=1024.937,202.676,-117.338,168.993,47.651,158.996
C06141=1024.943,202.925,-117.363,168.997,47.647,158.996
C06142=1024.949,203.173,-117.387,169.002,47.643,158.995
C06143=1024.955,203.422,-117.411,169.006,47.639,158.995
C06144=1024.978,204.455,-117.512,169.408,47.739,159.070
C06145=1024.990,204.861,-117.554,169.413,47.733,159.069
C06146=1025.000,205.266,-117.596,169.418,47.728,159.069
C06147=1025.011,205.671,-117.638,169.422,47.723,159.068
C06148=1025.021,206.078,-117.681,169.428,47.717,159.068
C06149=1025.028,206.326,-117.707,169.431,47.714,159.068
C06150=1025.034,206.575,-117.733,169.434,47.710,159.067
C06151=1025.041,206.823,-117.759,169.438,47.706,159.067
C06152=1025.048,207.071,-117.785,169.441,47.703,159.067
C06153=1025.054,207.321,-117.811,169.444,47.700,159.067
C06154=1025.061,207.569,-117.837,169.447,47.697,159.066
C06155=1025.067,207.817,-117.862,169.450,47.693,159.066
C06156=1025.074,208.066,-117.888,169.453,47.690,159.066
C06157=1025.080,208.314,-117.915,169.456,47.687,159.065
C06158=1025.086,208.563,-117.940,169.459,47.683,159.065
C06159=1025.093,208.812,-117.967,169.463,47.680,159.065
C06160=1025.100,209.060,-117.993,169.466,47.676,159.064
C06161=1025.106,209.308,-118.019,169.469,47.673,159.064
C06162=1025.112,209.558,-118.045,169.472,47.670,159.064
C06163=1025.119,209.806,-118.071,169.475,47.666,159.064
C06164=1025.126,210.054,-118.098,169.478,47.663,159.063
C06165=1025.132,210.303,-118.123,169.481,47.660,159.063
C06166=1025.139,210.551,-118.149,169.485,47.657,159.063
C06167=1025.145,210.800,-118.176,169.488,47.653,159.062
C06168=1025.152,211.048,-118.202,169.491,47.650,159.062
C06169=1025.158,211.297,-118.229,169.494,47.647,159.062
C06170=1025.164,211.545,-118.255,169.497,47.644,159.062
C06171=1025.171,211.794,-118.280,169.500,47.641,159.061
C06172=1025.177,212.043,-118.307,169.503,47.637,159.061
C06173=1025.184,212.291,-118.334,169.506,47.634,159.061
C06174=1025.190,212.540,-118.361,169.509,47.631,159.061
C06175=1025.196,212.788,-118.387,169.513,47.628,159.060
C06176=1025.203,213.036,-118.413,169.516,47.624,159.060
C06177=1025.209,213.285,-118.440,169.520,47.621,159.060
C06178=1025.216,213.533,-118.466,169.523,47.618,159.060
C06179=1025.223,213.782,-118.492,169.526,47.615,159.059
C06180=1025.229,214.030,-118.519,169.529,47.611,159.059
C06181=1025.236,214.279,-118.545,169.532,47.608,159.059
C06182=1025.242,214.528,-118.572,169.535,47.605,159.058
C06183=1025.248,214.777,-118.598,169.538,47.602,159.058
C06184=1025.255,215.025,-118.624,169.542,47.599,159.058
C06185=1025.261,215.274,-118.651,169.545,47.596,159.058
C06186=1025.268,215.522,-118.677,169.548,47.593,159.058
C06187=1025.274,215.771,-118.704,169.551,47.590,159.057
C06188=1025.281,216.019,-118.730,169.554,47.587,159.057
C06189=1025.288,216.268,-118.756,169.558,47.583,159.057
C06190=1025.294,216.516,-118.783,169.560,47.580,159.056
C06191=1025.301,216.765,-118.809,169.564,47.576,159.056
C06192=1025.307,217.013,-118.837,169.568,47.573,159.056
C06193=1025.314,217.262,-118.863,169.571,47.570,159.056
C06194=1025.320,217.510,-118.889,169.574,47.567,159.056
C06195=1025.327,217.759,-118.916,169.577,47.564,159.055
C06196=1025.333,218.007,-118.942,169.580,47.561,159.055
C06197=1025.340,218.256,-118.969,169.583,47.558,159.055
C06198=1025.346,218.504,-118.995,169.587,47.555,159.055
C06199=1025.353,218.753,-119.022,169.590,47.551,159.054
C06200=1025.359,219.001,-119.048,169.593,47.548,159.054
C06201=1025.371,219.409,-119.093,169.599,47.543,159.054
C06202=1025.381,219.818,-119.138,169.604,47.539,159.053
C06203=1025.391,220.226,-119.181,169.609,47.534,159.053
C06204=1025.402,220.634,-119.225,169.615,47.528,159.053
C06205=1025.408,220.882,-119.252,169.618,47.525,159.052
C06206=1025.414,221.131,-119.279,169.621,47.523,159.052
C06207=1025.421,221.379,-119.306,169.624,47.520,159.052
C06208=1025.427,221.628,-119.333,169.628,47.517,159.052
C06209=1025.434,221.877,-119.360,169.631,47.514,159.052
C06210=1025.441,222.124,-119.386,169.634,47.511,159.051
C06211=1025.447,222.373,-119.413,169.638,47.507,159.051
C06212=1025.453,222.622,-119.440,169.641,47.505,159.051
C06213=1025.460,222.870,-119.467,169.644,47.502,159.051
C06214=1025.467,223.119,-119.494,169.648,47.499,159.051
C06215=1025.473,223.367,-119.522,169.651,47.496,159.050
C06216=1025.479,223.616,-119.549,169.654,47.493,159.050
C06217=1025.486,223.864,-119.575,169.657,47.490,159.050
C06218=1025.492,224.112,-119.602,169.660,47.487,159.050
C06219=1025.499,224.361,-119.629,169.664,47.484,159.050
C06220=1025.505,224.609,-119.656,169.668,47.481,159.049
C06221=1025.512,224.858,-119.683,169.671,47.478,159.049
C06222=1025.518,225.107,-119.710,169.674,47.475,159.049
C06223=1025.525,225.354,-119.737,169.677,47.472,159.049
C06224=1025.531,225.603,-119.764,169.680,47.469,159.049
C06225=1025.538,225.852,-119.792,169.684,47.467,159.048
C06226=1025.544,226.101,-119.819,169.688,47.463,159.048
C06227=1025.551,226.348,-119.845,169.691,47.460,159.048
C06228=1025.558,226.597,-119.872,169.694,47.457,159.048
C06229=1025.564,226.846,-119.900,169.698,47.455,159.048
C06230=1025.571,227.094,-119.926,169.701,47.452,159.047
C06231=1025.578,227.342,-119.954,169.704,47.449,159.047
C06232=1025.584,227.591,-119.982,169.707,47.446,159.047
C06233=1025.590,227.839,-120.008,169.710,47.443,159.047
C06234=1025.597,228.088,-120.036,169.714,47.440,159.047
C06235=1025.603,228.337,-120.063,169.718,47.438,159.047
C06236=1025.610,228.585,-120.091,169.721,47.434,159.046
C06237=1025.616,228.833,-120.118,169.724,47.432,159.046
C06238=1025.622,229.082,-120.145,169.728,47.429,159.046
C06239=1025.629,229.330,-120.173,169.731,47.427,159.046
C06240=1025.635,229.578,-120.200,169.734,47.424,159.046
C06241=1025.642,229.827,-120.228,169.737,47.420,159.046
C06242=1025.649,230.075,-120.254,169.741,47.418,159.045
C06243=1025.655,230.324,-120.282,169.745,47.415,159.045
C06244=1025.661,230.571,-120.310,169.748,47.412,159.045
C06245=1025.668,230.820,-120.337,169.751,47.409,159.045
C06246=1025.675,231.069,-120.364,169.755,47.407,159.045
C06247=1025.680,231.318,-120.393,169.758,47.404,159.045
C06248=1025.687,231.565,-120.420,169.761,47.401,159.045
C06249=1025.693,231.814,-120.448,169.765,47.399,159.044
C06250=1025.700,232.062,-120.475,169.768,47.396,159.044
C06251=1025.706,232.311,-120.502,169.771,47.394,159.044
C06252=1025.713,232.560,-120.530,169.775,47.390,159.044
C06253=1025.719,232.808,-120.558,169.779,47.388,159.044
C06254=1025.726,233.056,-120.585,169.782,47.385,159.044
C06255=1025.732,233.304,-120.613,169.785,47.382,159.044
C06256=1025.739,233.553,-120.641,169.789,47.380,159.043
C06257=1025.749,233.953,-120.686,169.795,47.375,159.043
C06258=1025.760,234.354,-120.730,169.799,47.371,159.043
C06259=1025.770,234.754,-120.775,169.805,47.367,159.043
C06260=1025.780,235.155,-120.819,169.811,47.362,159.043
C06261=1025.786,235.403,-120.847,169.815,47.360,159.042
C06262=1025.793,235.652,-120.875,169.818,47.357,159.042
C06263=1025.800,235.900,-120.902,169.821,47.354,159.042
C06264=1025.806,236.149,-120.930,169.825,47.352,159.042
C06265=1025.813,236.397,-120.958,169.828,47.349,159.042
C06266=1025.820,236.645,-120.986,169.832,47.346,159.042
C06267=1025.826,236.893,-121.014,169.835,47.344,159.042
C06268=1025.833,237.141,-121.041,169.839,47.341,159.042
C06269=1025.839,237.390,-121.070,169.842,47.338,159.041
C06270=1025.846,237.638,-121.097,169.845,47.336,159.041
C06271=1025.852,237.887,-121.125,169.849,47.334,159.041
C06272=1025.859,238.135,-121.153,169.852,47.330,159.041
C06273=1025.866,238.384,-121.181,169.856,47.328,159.041
C06274=1025.871,238.632,-121.209,169.860,47.325,159.041
C06275=1025.878,238.881,-121.237,169.863,47.323,159.041
C06276=1025.885,239.129,-121.265,169.866,47.320,159.041
C06277=1025.892,239.377,-121.293,169.870,47.318,159.041
C06278=1025.899,239.625,-121.321,169.873,47.315,159.040
C06279=1025.904,239.874,-121.349,169.877,47.313,159.040
C06280=1025.911,240.122,-121.376,169.881,47.310,159.040
C06281=1025.918,240.370,-121.405,169.885,47.308,159.040
C06282=1025.923,240.619,-121.433,169.888,47.305,159.040
C06283=1025.930,240.867,-121.461,169.891,47.302,159.040
C06284=1025.936,241.115,-121.490,169.895,47.300,159.040
C06285=1025.943,241.364,-121.518,169.898,47.297,159.040
C06286=1025.949,241.612,-121.546,169.901,47.295,159.040
C06287=1025.956,241.860,-121.574,169.905,47.293,159.040
C06288=1025.963,242.109,-121.602,169.909,47.290,159.040
C06289=1025.969,242.357,-121.631,169.913,47.288,159.040
C06290=1025.976,242.605,-121.659,169.916,47.285,159.039
C06291=1025.982,242.854,-121.687,169.920,47.283,159.039
C06292=1025.989,243.102,-121.716,169.923,47.280,159.039
C06293=1025.995,243.350,-121.744,169.926,47.278,159.039
C06294=1026.001,243.598,-121.772,169.930,47.276,159.039
C06295=1026.007,243.847,-121.801,169.933,47.273,159.039
C06296=1026.014,244.095,-121.829,169.938,47.271,159.039
C06297=1026.020,244.344,-121.858,169.941,47.268,159.039
C06298=1026.027,244.592,-121.887,169.945,47.266,159.039
C06299=1026.033,244.840,-121.914,169.948,47.263,159.039
C06300=1026.040,245.088,-121.943,169.951,47.261,159.039
C06301=1026.046,245.336,-121.972,169.955,47.259,159.039
C06302=1026.052,245.585,-122.000,169.958,47.256,159.039
C06303=1026.059,245.833,-122.029,169.962,47.255,159.039
C06304=1026.065,246.082,-122.057,169.966,47.252,159.039
C06305=1026.071,246.330,-122.087,169.970,47.249,159.039
C06306=1026.078,246.578,-122.115,169.973,47.247,159.039
C06307=1026.084,246.826,-122.143,169.977,47.245,159.038
C06308=1026.090,247.075,-122.172,169.980,47.242,159.038
C06309=1026.097,247.322,-122.201,169.984,47.241,159.038
C06310=1026.103,247.571,-122.229,169.987,47.238,159.038
C06311=1026.109,247.819,-122.258,169.991,47.236,159.038
C06312=1026.116,248.067,-122.287,169.994,47.233,159.038
C06313=1026.126,248.462,-122.333,170.000,47.230,159.038
C06314=1026.136,248.856,-122.379,170.007,47.226,159.038
C06315=1026.147,249.251,-122.424,170.012,47.223,159.038
C06316=1026.157,249.644,-122.470,170.018,47.219,159.038
C06317=1026.163,249.893,-122.498,170.022,47.217,159.038
C06318=1026.170,250.141,-122.527,170.025,47.214,159.038
C06319=1026.177,250.390,-122.556,170.028,47.212,159.038
C06320=1026.183,250.638,-122.585,170.032,47.210,159.038
C06321=1026.189,250.886,-122.614,170.036,47.208,159.038
C06322=1026.196,251.134,-122.643,170.040,47.205,159.038
C06323=1026.202,251.382,-122.671,170.044,47.203,159.038
C06324=1026.209,251.631,-122.700,170.047,47.201,159.038
C06325=1026.215,251.879,-122.729,170.051,47.199,159.038
C06326=1026.222,252.127,-122.758,170.054,47.196,159.038
C06327=1026.228,252.375,-122.787,170.058,47.194,159.038
C06328=1026.235,252.624,-122.816,170.062,47.192,159.038
C06329=1026.241,252.872,-122.845,170.066,47.189,159.038
C06330=1026.248,253.120,-122.874,170.069,47.188,159.038
C06331=1026.255,253.368,-122.903,170.073,47.185,159.038
C06332=1026.261,253.616,-122.932,170.076,47.183,159.038
C06333=1026.267,253.865,-122.961,170.081,47.181,159.038
C06334=1026.275,254.113,-122.990,170.085,47.178,159.038
C06335=1026.281,254.361,-123.019,170.088,47.176,159.038
C06336=1026.287,254.609,-123.048,170.092,47.174,159.038
C06337=1026.294,254.858,-123.077,170.095,47.172,159.038
C06338=1026.301,255.106,-123.106,170.100,47.169,159.038
C06339=1026.307,255.354,-123.135,170.103,47.168,159.038
C06340=1026.314,255.602,-123.164,170.107,47.165,159.038
C06341=1026.320,255.851,-123.193,170.110,47.163,159.038
C06342=1026.327,256.099,-123.222,170.114,47.161,159.038
C06343=1026.334,256.347,-123.251,170.118,47.158,159.038
C06344=1026.341,256.596,-123.280,170.122,47.157,159.038
C06345=1026.347,256.844,-123.309,170.126,47.154,159.038
C06346=1026.354,257.092,-123.337,170.129,47.153,159.038
C06347=1026.361,257.341,-123.367,170.133,47.150,159.038
C06348=1026.367,257.588,-123.397,170.137,47.148,159.038
C06349=1026.373,257.836,-123.426,170.141,47.146,159.038
C06350=1026.380,258.085,-123.455,170.145,47.144,159.038
C06351=1026.387,258.333,-123.484,170.148,47.142,159.038
C06352=1026.394,258.581,-123.513,170.152,47.139,159.038
C06353=1026.400,258.830,-123.542,170.156,47.137,159.038
C06354=1026.407,259.077,-123.572,170.160,47.135,159.038
C06355=1026.415,259.326,-123.601,170.163,47.133,159.038
C06356=1026.421,259.574,-123.630,170.168,47.131,159.038
C06357=1026.427,259.822,-123.659,170.172,47.129,159.038
C06358=1026.434,260.070,-123.689,170.175,47.127,159.038
C06359=1026.441,260.318,-123.717,170.179,47.125,159.038
C06360=1026.448,260.567,-123.747,170.183,47.122,159.038
C06361=1026.454,260.815,-123.776,170.187,47.120,159.038
C06362=1026.461,261.063,-123.805,170.191,47.119,159.038
C06363=1026.468,261.312,-123.835,170.194,47.116,159.038
C06364=1026.474,261.559,-123.865,170.198,47.115,159.038
C06365=1026.480,261.808,-123.895,170.203,47.113,159.038
C06366=1026.487,262.056,-123.924,170.206,47.111,159.038
C06367=1026.493,262.304,-123.953,170.210,47.108,159.038
C06368=1026.500,262.552,-123.983,170.213,47.107,159.038
C06369=1026.510,262.945,-124.031,170.220,47.104,159.038
C06370=1026.521,263.338,-124.078,170.226,47.100,159.039
C06371=1026.531,263.730,-124.124,170.232,47.097,159.039
C06372=1026.542,264.123,-124.171,170.238,47.094,159.039
C06373=1026.548,264.371,-124.201,170.242,47.093,159.039
C06374=1026.555,264.619,-124.231,170.246,47.091,159.039
C06375=1026.561,264.868,-124.261,170.251,47.089,159.039
C06376=1026.568,265.116,-124.291,170.254,47.086,159.039
C06377=1026.575,265.363,-124.320,170.258,47.085,159.039
C06378=1026.581,265.612,-124.350,170.261,47.083,159.039
C06379=1026.587,265.860,-124.380,170.265,47.081,159.039
C06380=1026.595,266.108,-124.410,170.270,47.079,159.039
C06381=1026.601,266.356,-124.439,170.274,47.078,159.040
C06382=1026.607,266.605,-124.470,170.277,47.076,159.040
C06383=1026.614,266.852,-124.500,170.281,47.074,159.040
C06384=1026.621,267.100,-124.530,170.286,47.072,159.040
C06385=1026.627,267.348,-124.560,170.289,47.070,159.040
C06386=1026.634,267.597,-124.590,170.293,47.068,159.040
C06387=1026.640,267.845,-124.619,170.297,47.066,159.040
C06388=1026.647,268.093,-124.650,170.302,47.064,159.040
C06389=1026.653,268.341,-124.680,170.305,47.063,159.040
C06390=1026.660,268.589,-124.710,170.309,47.061,159.040
C06391=1026.666,268.837,-124.740,170.313,47.059,159.040
C06392=1026.673,269.085,-124.770,170.318,47.057,159.041
C06393=1026.680,269.334,-124.800,170.321,47.055,159.041
C06394=1026.686,269.582,-124.830,170.325,47.054,159.041
C06395=1026.693,269.830,-124.860,170.329,47.052,159.041
C06396=1026.700,270.077,-124.890,170.333,47.050,159.041
C06397=1026.706,270.326,-124.921,170.337,47.048,159.041
C06398=1026.713,270.574,-124.951,170.341,47.046,159.041
C06399=1026.719,270.822,-124.981,170.345,47.045,159.041
C06400=1026.726,271.070,-125.011,170.350,47.043,159.042
C06401=1026.732,271.318,-125.042,170.353,47.042,159.042
C06402=1026.739,271.566,-125.072,170.357,47.040,159.042
C06403=1026.746,271.814,-125.103,170.361,47.038,159.042
C06404=1026.752,272.062,-125.133,170.366,47.036,159.042
C06405=1026.759,272.310,-125.164,170.369,47.035,159.042
C06406=1026.766,272.558,-125.194,170.373,47.033,159.042
C06407=1026.772,272.806,-125.224,170.377,47.032,159.042
C06408=1026.779,273.054,-125.254,170.382,47.030,159.043
C06409=1026.785,273.303,-125.285,170.386,47.028,159.043
C06410=1026.792,273.550,-125.316,170.389,47.026,159.043
C06411=1026.799,273.798,-125.346,170.393,47.025,159.043
C06412=1026.805,274.047,-125.377,170.398,47.023,159.043
C06413=1026.812,274.294,-125.407,170.402,47.021,159.043
C06414=1026.818,274.543,-125.438,170.406,47.020,159.043
C06415=1026.825,274.791,-125.469,170.410,47.019,159.044
C06416=1026.831,275.038,-125.499,170.414,47.017,159.044
C06417=1026.838,275.287,-125.529,170.418,47.015,159.044
C06418=1026.845,275.534,-125.560,170.422,47.013,159.044
C06419=1026.852,275.783,-125.591,170.427,47.012,159.044
C06420=1026.858,276.031,-125.621,170.431,47.010,159.044
C06421=1026.865,276.278,-125.652,170.434,47.008,159.044
C06422=1026.871,276.527,-125.683,170.439,47.007,159.045
C06423=1026.879,276.775,-125.713,170.443,47.005,159.045
C06424=1026.885,277.022,-125.744,170.447,47.004,159.045
C06425=1026.896,277.420,-125.794,170.454,47.001,159.045
C06426=1026.906,277.818,-125.843,170.461,46.999,159.046
C06427=1026.916,278.215,-125.892,170.467,46.996,159.046
C06428=1026.928,278.612,-125.942,170.474,46.994,159.046
C06429=1026.933,278.860,-125.972,170.478,46.992,159.046
C06430=1026.940,279.108,-126.004,170.482,46.991,159.047
C06431=1026.947,279.356,-126.035,170.486,46.990,159.047
C06432=1026.953,279.604,-126.066,170.491,46.988,159.047
C06433=1026.960,279.852,-126.097,170.495,46.987,159.047
C06434=1026.967,280.100,-126.127,170.499,46.986,159.047
C06435=1026.973,280.348,-126.158,170.503,46.984,159.048
C06436=1026.980,280.596,-126.190,170.507,46.982,159.048
C06437=1026.986,280.844,-126.221,170.511,46.981,159.048
C06438=1026.993,281.092,-126.252,170.516,46.979,159.048
C06439=1027.000,281.340,-126.283,170.520,46.978,159.048
C06440=1027.006,281.588,-126.314,170.524,46.977,159.049
C06441=1027.012,281.836,-126.345,170.528,46.976,159.049
C06442=1027.020,282.083,-126.376,170.533,46.974,159.049
C06443=1027.027,282.331,-126.408,170.537,46.972,159.049
C06444=1027.033,282.580,-126.438,170.541,46.971,159.049
C06445=1027.040,282.828,-126.470,170.546,46.969,159.050
C06446=1027.047,283.075,-126.501,170.550,46.968,159.050
C06447=1027.053,283.323,-126.533,170.553,46.967,159.050
C06448=1027.060,283.571,-126.564,170.558,46.965,159.050
C06449=1027.067,283.820,-126.594,170.563,46.964,159.051
C06450=1027.074,284.067,-126.626,170.567,46.962,159.051
C06451=1027.081,284.315,-126.657,170.571,46.961,159.051
C06452=1027.087,284.563,-126.688,170.575,46.960,159.051
C06453=1027.094,284.811,-126.720,170.580,46.958,159.051
C06454=1027.101,285.059,-126.751,170.584,46.957,159.052
C06455=1027.107,285.307,-126.783,170.588,46.956,159.052
C06456=1027.114,285.555,-126.814,170.593,46.954,159.052
C06457=1027.121,285.803,-126.846,170.597,46.953,159.052
C06458=1027.128,286.051,-126.877,170.601,46.952,159.053
C06459=1027.134,286.299,-126.908,170.606,46.950,159.053
C06460=1027.141,286.546,-126.940,170.610,46.949,159.053
C06461=1027.148,286.794,-126.971,170.615,46.947,159.053
C06462=1027.155,287.042,-127.003,170.619,46.946,159.054
C06463=1027.161,287.290,-127.034,170.623,46.945,159.054
C06464=1027.168,287.538,-127.066,170.628,46.944,159.054
C06465=1027.175,287.786,-127.097,170.632,46.943,159.054
C06466=1027.181,288.034,-127.128,170.636,46.942,159.055
C06467=1027.188,288.282,-127.160,170.641,46.940,159.055
C06468=1027.194,288.529,-127.193,170.645,46.939,159.055
C06469=1027.201,288.777,-127.224,170.649,46.938,159.056
C06470=1027.208,289.025,-127.255,170.654,46.936,159.056
C06471=1027.215,289.273,-127.287,170.658,46.935,159.056
C06472=1027.222,289.520,-127.319,170.663,46.934,159.056
C06473=1027.228,289.769,-127.351,170.667,46.933,159.057
C06474=1027.234,290.016,-127.383,170.671,46.932,159.057
C06475=1027.241,290.264,-127.414,170.676,46.930,159.057
C06476=1027.249,290.512,-127.446,170.680,46.929,159.057
C06477=1027.255,290.760,-127.478,170.685,46.928,159.058
C06478=1027.262,291.008,-127.509,170.689,46.927,159.058
C06479=1027.268,291.256,-127.542,170.693,46.926,159.058
C06480=1027.275,291.504,-127.574,170.698,46.924,159.059
C06481=1027.287,291.914,-127.626,170.706,46.923,159.059
C06482=1027.297,292.323,-127.679,170.713,46.921,159.060
C06483=1027.309,292.732,-127.732,170.721,46.919,159.060
C06484=1027.320,293.142,-127.785,170.728,46.917,159.061
C06485=1027.327,293.390,-127.817,170.732,46.916,159.061
C06486=1027.334,293.638,-127.849,170.737,46.915,159.061
C06487=1027.340,293.885,-127.881,170.741,46.914,159.062
C06488=1027.347,294.133,-127.913,170.746,46.913,159.062
C06489=1027.353,294.381,-127.946,170.750,46.912,159.062
C06490=1027.361,294.629,-127.978,170.754,46.911,159.062
C06491=1027.367,294.877,-128.010,170.760,46.910,159.063
C06492=1027.373,295.124,-128.043,170.764,46.909,159.063
C06493=1027.380,295.372,-128.075,170.769,46.908,159.064
C06494=1027.387,295.619,-128.108,170.773,46.907,159.064
C06495=1027.393,295.868,-128.140,170.777,46.906,159.064
C06496=1027.400,296.116,-128.172,170.783,46.905,159.065
C06497=1027.406,296.363,-128.205,170.787,46.904,159.065
C06498=1027.414,296.610,-128.237,170.792,46.903,159.065
C06499=1027.420,296.858,-128.270,170.796,46.902,159.066
C06500=1027.426,297.107,-128.302,170.800,46.901,159.066
C06501=1027.433,297.354,-128.335,170.805,46.901,159.066
C06502=1027.440,297.602,-128.367,170.809,46.900,159.067
C06503=1027.447,297.850,-128.400,170.814,46.898,159.067
C06504=1027.454,298.097,-128.433,170.819,46.898,159.068
C06505=1027.460,298.345,-128.465,170.824,46.896,159.068
C06506=1027.466,298.593,-128.498,170.828,46.896,159.068
C06507=1027.474,298.841,-128.531,170.832,46.895,159.069
C06508=1027.480,299.088,-128.563,170.838,46.894,159.069
C06509=1027.486,299.336,-128.596,170.842,46.893,159.069
C06510=1027.494,299.584,-128.629,170.847,46.892,159.070
C06511=1027.500,299.831,-128.661,170.851,46.891,159.070
C06512=1027.507,300.080,-128.694,170.856,46.891,159.071
C06513=1027.514,300.327,-128.727,170.860,46.890,159.071
C06514=1027.521,300.574,-128.759,170.866,46.889,159.071
C06515=1027.527,300.823,-128.792,170.870,46.888,159.072
C06516=1027.535,301.070,-128.825,170.875,46.887,159.072
C06517=1027.541,301.318,-128.857,170.879,46.887,159.072
C06518=1027.548,301.566,-128.890,170.884,46.885,159.073
C06519=1027.555,301.813,-128.923,170.889,46.885,159.073
C06520=1027.562,302.061,-128.956,170.894,46.884,159.074
C06521=1027.568,302.308,-128.989,170.898,46.883,159.074
C06522=1027.576,302.556,-129.022,170.904,46.882,159.074
C06523=1027.582,302.804,-129.054,170.908,46.881,159.075
C06524=1027.589,303.052,-129.087,170.913,46.880,159.075
C06525=1027.596,303.299,-129.121,170.917,46.880,159.076
C06526=1027.603,303.547,-129.153,170.922,46.879,159.076
C06527=1027.610,303.795,-129.186,170.927,46.878,159.076
C06528=1027.616,304.043,-129.219,170.932,46.878,159.077
C06529=1027.624,304.290,-129.252,170.936,46.877,159.077
C06530=1027.631,304.538,-129.285,170.941,46.876,159.078
C06531=1027.637,304.786,-129.318,170.946,46.875,159.078
C06532=1027.645,305.033,-129.351,170.951,46.875,159.079
C06533=1027.651,305.281,-129.384,170.955,46.873,159.079
C06534=1027.658,305.529,-129.417,170.960,46.873,159.079
C06535=1027.665,305.776,-129.450,170.966,46.872,159.080
C06536=1027.672,306.024,-129.483,170.970,46.872,159.080
C06537=1027.679,306.237,-129.512,170.974,46.871,159.081
C06538=1027.684,306.451,-129.541,170.978,46.870,159.081
C06539=1027.690,306.664,-129.569,170.983,46.870,159.081
C06540=1027.696,306.877,-129.598,170.987,46.869,159.082
C06541=1027.703,307.091,-129.626,170.991,46.868,159.082
C06542=1027.709,307.304,-129.654,170.995,46.868,159.083
C06543=1027.715,307.518,-129.683,171.000,46.867,159.083
C06544=1027.721,307.731,-129.711,171.004,46.866,159.083
C06545=1027.728,307.978,-129.745,171.008,46.866,159.084
C06546=1027.734,308.226,-129.778,171.014,46.865,159.084
C06547=1027.742,308.474,-129.811,171.019,46.864,159.085
C06548=1027.749,308.721,-129.844,171.023,46.864,159.085
C06549=1027.756,308.969,-129.878,171.029,46.863,159.086
C06550=1027.764,309.216,-129.911,171.033,46.863,159.086
C06551=1027.771,309.465,-129.944,171.038,46.862,159.087
C06552=1027.777,309.712,-129.978,171.044,46.861,159.087
C06553=1027.784,309.959,-130.011,171.048,46.861,159.087
C06554=1027.792,310.207,-130.044,171.053,46.860,159.088
C06555=1027.799,310.455,-130.078,171.059,46.859,159.088
C06556=1027.806,310.702,-130.111,171.063,46.859,159.089
C06557=1027.813,310.950,-130.144,171.068,46.858,159.089
C06558=1027.820,311.198,-130.178,171.073,46.858,159.090
C06559=1027.827,311.445,-130.212,171.078,46.857,159.090
C06560=1027.833,311.693,-130.246,171.083,46.856,159.091
C06561=1027.840,311.941,-130.280,171.088,46.856,159.091
C06562=1027.847,312.188,-130.313,171.093,46.856,159.092
C06563=1027.854,312.435,-130.347,171.098,46.855,159.092
C06564=1027.861,312.683,-130.382,171.103,46.854,159.093
C06565=1027.868,312.931,-130.415,171.108,46.855,159.093
C06566=1027.875,313.177,-130.450,171.113,46.854,159.094
C06567=1027.881,313.425,-130.484,171.118,46.853,159.094
C06568=1027.888,313.673,-130.518,171.123,46.853,159.095
C06569=1027.895,313.921,-130.552,171.128,46.853,159.096
C06570=1027.902,314.169,-130.586,171.134,46.852,159.096
C06571=1027.909,314.416,-130.620,171.138,46.852,159.097
C06572=1027.916,314.663,-130.653,171.144,46.851,159.097
C06573=1027.923,314.911,-130.688,171.148,46.852,159.098
C06574=1027.930,315.158,-130.722,171.154,46.851,159.098
C06575=1027.937,315.406,-130.756,171.159,46.850,159.099
C06576=1027.943,315.654,-130.791,171.164,46.850,159.099
C06577=1027.950,315.901,-130.824,171.169,46.850,159.100
C06578=1027.957,316.148,-130.859,171.174,46.849,159.101
C06579=1027.964,316.396,-130.893,171.179,46.849,159.101
C06580=1027.971,316.644,-130.927,171.184,46.849,159.102
C06581=1027.978,316.891,-130.962,171.190,46.848,159.102
C06582=1027.985,317.139,-130.996,171.194,46.848,159.103
C06583=1027.992,317.386,-131.030,171.200,46.848,159.103
C06584=1027.999,317.634,-131.065,171.205,46.848,159.104
C06585=1028.006,317.881,-131.099,171.210,46.847,159.104
C06586=1028.014,318.128,-131.133,171.215,46.847,159.105
C06587=1028.020,318.376,-131.167,171.221,46.846,159.105
C06588=1028.027,318.624,-131.201,171.225,46.846,159.106
C06589=1028.035,318.871,-131.236,171.231,46.846,159.107
C06590=1028.041,319.119,-131.270,171.236,46.846,159.107
C06591=1028.049,319.366,-131.305,171.241,46.846,159.108
C06592=1028.055,319.614,-131.339,171.246,46.845,159.108
C06593=1028.063,319.861,-131.374,171.252,46.845,159.109
C06594=1028.070,320.109,-131.408,171.258,46.845,159.110
C06595=1028.077,320.356,-131.443,171.262,46.844,159.110
C06596=1028.084,320.604,-131.477,171.268,46.844,159.111
C06597=1028.091,320.820,-131.507,171.272,46.844,159.111
C06598=1028.097,321.036,-131.537,171.277,46.844,159.112
C06599=1028.103,321.252,-131.567,171.282,46.843,159.112
C06600=1028.109,321.468,-131.597,171.287,46.843,159.113
C06601=1028.115,321.683,-131.627,171.291,46.843,159.113
C06602=1028.122,321.900,-131.658,171.296,46.843,159.114
C06603=1028.128,322.114,-131.688,171.300,46.843,159.114
C06604=1028.134,322.331,-131.719,171.304,46.843,159.115
C06605=1028.142,322.579,-131.752,171.310,46.843,159.116
C06606=1028.149,322.826,-131.787,171.315,46.842,159.116
C06607=1028.156,323.074,-131.822,171.321,46.842,159.117
C06608=1028.164,323.321,-131.856,171.326,46.842,159.117
C06609=1028.170,323.569,-131.891,171.331,46.842,159.118
C06610=1028.178,323.816,-131.926,171.337,46.842,159.119
C06611=1028.185,324.063,-131.960,171.343,46.842,159.120
C06612=1028.193,324.311,-131.996,171.348,46.841,159.120
C06613=1028.200,324.558,-132.030,171.354,46.841,159.121
C06614=1028.207,324.806,-132.065,171.358,46.841,159.121
C06615=1028.215,325.054,-132.100,171.364,46.841,159.122
C06616=1028.222,325.301,-132.134,171.370,46.841,159.123
C06617=1028.229,325.548,-132.169,171.375,46.841,159.123
C06618=1028.237,325.795,-132.204,171.381,46.841,159.124
C06619=1028.244,326.043,-132.240,171.386,46.840,159.125
C06620=1028.252,326.290,-132.274,171.391,46.841,159.125
C06621=1028.260,326.538,-132.309,171.397,46.841,159.126
C06622=1028.266,326.785,-132.344,171.402,46.840,159.127
C06623=1028.274,327.032,-132.379,171.408,46.840,159.127
C06624=1028.281,327.280,-132.414,171.414,46.840,159.128
C06625=1028.289,327.528,-132.449,171.419,46.840,159.129
C06626=1028.296,327.775,-132.484,171.425,46.840,159.129
C06627=1028.303,328.023,-132.519,171.430,46.840,159.130
C06628=1028.311,328.269,-132.555,171.435,46.840,159.131
C06629=1028.318,328.517,-132.590,171.441,46.841,159.131
C06630=1028.325,328.765,-132.625,171.447,46.840,159.132
C06631=1028.332,329.012,-132.661,171.452,46.840,159.133
C06632=1028.339,329.260,-132.697,171.458,46.840,159.133
C06633=1028.346,329.507,-132.732,171.463,46.841,159.134
C06634=1028.353,329.754,-132.768,171.469,46.841,159.135
C06635=1028.361,330.002,-132.802,171.474,46.841,159.136
C06636=1028.368,330.249,-132.838,171.480,46.841,159.136
C06637=1028.376,330.496,-132.874,171.486,46.841,159.137
C06638=1028.383,330.744,-132.909,171.492,46.841,159.138
C06639=1028.390,330.991,-132.945,171.497,46.842,159.139
C06640=1028.397,331.238,-132.980,171.503,46.841,159.139
C06641=1028.405,331.486,-133.016,171.509,46.841,159.140
C06642=1028.412,331.733,-133.051,171.514,46.842,159.141
C06643=1028.420,331.980,-133.087,171.519,46.842,159.141
C06644=1028.427,332.228,-133.122,171.525,46.842,159.142
C06645=1028.434,332.475,-133.159,171.531,46.842,159.143
C06646=1028.441,332.723,-133.194,171.537,46.843,159.144
C06647=1028.449,332.970,-133.230,171.543,46.843,159.144
C06648=1028.457,333.217,-133.266,171.548,46.843,159.145
C06649=1028.464,333.465,-133.301,171.554,46.843,159.146
C06650=1028.472,333.712,-133.337,171.560,46.844,159.147
C06651=1028.479,333.959,-133.373,171.566,46.843,159.148
C06652=1028.486,334.206,-133.409,171.572,46.844,159.148
C06653=1028.494,334.454,-133.445,171.577,46.844,159.149
C06654=1028.501,334.701,-133.480,171.583,46.844,159.150
C06655=1028.508,334.948,-133.517,171.589,46.845,159.151
C06656=1028.515,335.195,-133.553,171.595,46.845,159.151
C06657=1028.522,335.410,-133.584,171.600,46.846,159.152
C06658=1028.528,335.623,-133.615,171.604,46.846,159.153
C06659=1028.534,335.837,-133.646,171.609,46.846,159.153
C06660=1028.541,336.050,-133.678,171.615,46.846,159.154
C06661=1028.547,336.264,-133.709,171.620,46.846,159.155
C06662=1028.554,336.477,-133.740,171.624,46.847,159.156
C06663=1028.560,336.691,-133.772,171.630,46.847,159.156
C06664=1028.566,336.905,-133.803,171.635,46.847,159.157
C06665=1028.574,337.152,-133.839,171.641,46.848,159.158
C06666=1028.581,337.399,-133.875,171.647,46.848,159.159
C06667=1028.589,337.646,-133.911,171.653,46.849,159.160
C06668=1028.597,337.894,-133.947,171.659,46.849,159.160
C06669=1028.603,338.142,-133.984,171.664,46.849,159.161
C06670=1028.611,338.388,-134.020,171.670,46.850,159.162
C06671=1028.618,338.636,-134.056,171.676,46.850,159.163
C06672=1028.626,338.883,-134.093,171.682,46.851,159.164
C06673=1028.634,339.130,-134.129,171.688,46.851,159.164
C06674=1028.642,339.377,-134.165,171.694,46.852,159.165
C06675=1028.649,339.625,-134.202,171.700,46.852,159.166
C06676=1028.656,339.872,-134.238,171.706,46.853,159.167
C06677=1028.664,340.119,-134.275,171.712,46.853,159.168
C06678=1028.671,340.366,-134.311,171.718,46.853,159.169
C06679=1028.679,340.614,-134.347,171.724,46.854,159.170
C06680=1028.687,340.860,-134.384,171.731,46.854,159.171
C06681=1028.694,341.108,-134.421,171.737,46.855,159.171
C06682=1028.702,341.355,-134.458,171.742,46.855,159.172
C06683=1028.709,341.603,-134.495,171.749,46.856,159.173
C06684=1028.716,341.849,-134.532,171.755,46.857,159.174
C06685=1028.724,342.096,-134.568,171.761,46.857,159.175
C06686=1028.731,342.343,-134.605,171.767,46.858,159.176
C06687=1028.739,342.591,-134.641,171.772,46.858,159.177
C06688=1028.747,342.838,-134.678,171.779,46.859,159.178
C06689=1028.754,343.086,-134.715,171.785,46.860,159.179
C06690=1028.762,343.332,-134.752,171.791,46.860,159.179
C06691=1028.769,343.579,-134.790,171.798,46.860,159.180
C06692=1028.777,343.827,-134.826,171.804,46.862,159.181
C06693=1028.784,344.074,-134.863,171.810,46.862,159.182
C06694=1028.792,344.321,-134.900,171.816,46.863,159.183
C06695=1028.799,344.568,-134.937,171.822,46.864,159.184
C06696=1028.807,344.815,-134.974,171.828,46.864,159.185
C06697=1028.815,345.062,-135.011,171.834,46.865,159.186
C06698=1028.822,345.309,-135.049,171.841,46.865,159.187
C06699=1028.830,345.556,-135.085,171.847,46.866,159.188
C06700=1028.837,345.805,-135.123,171.853,46.867,159.189
C06701=1028.845,346.052,-135.160,171.859,46.867,159.190
C06702=1028.853,346.299,-135.197,171.865,46.869,159.191
C06703=1028.861,346.546,-135.234,171.871,46.869,159.192
C06704=1028.868,346.793,-135.272,171.879,46.870,159.193
C06705=1028.876,347.039,-135.309,171.885,46.870,159.194
C06706=1028.883,347.287,-135.346,171.891,46.871,159.195
C06707=1028.892,347.534,-135.383,171.897,46.872,159.196
C06708=1028.899,347.781,-135.421,171.903,46.873,159.196
C06709=1028.907,348.028,-135.458,171.910,46.874,159.198
C06710=1028.915,348.275,-135.495,171.916,46.874,159.198
C06711=1028.922,348.522,-135.532,171.923,46.875,159.199
C06712=1028.930,348.770,-135.570,171.929,46.876,159.200
C06713=1028.938,349.016,-135.608,171.936,46.877,159.201
C06714=1028.945,349.263,-135.645,171.942,46.878,159.202
C06715=1028.953,349.510,-135.683,171.948,46.879,159.203
C06716=1028.961,349.758,-135.721,171.954,46.880,159.205
C06717=1028.967,349.970,-135.753,171.960,46.880,159.205
C06718=1028.974,350.181,-135.785,171.965,46.881,159.206
C06719=1028.981,350.393,-135.818,171.972,46.882,159.207
C06720=1028.987,350.606,-135.850,171.977,46.883,159.208
C06721=1028.994,350.817,-135.882,171.982,46.883,159.209
C06722=1029.001,351.030,-135.914,171.989,46.884,159.210
C06723=1029.007,351.242,-135.947,171.994,46.885,159.211
C06724=1029.014,351.454,-135.980,172.000,46.886,159.212
C06725=1029.021,351.701,-136.018,172.006,46.887,159.213
C06726=1029.029,351.947,-136.056,172.012,46.888,159.214
C06727=1029.038,352.195,-136.093,172.019,46.889,159.215
C06728=1029.045,352.441,-136.131,172.026,46.890,159.216
C06729=1029.053,352.689,-136.169,172.032,46.891,159.217
C06730=1029.060,352.936,-136.207,172.039,46.891,159.218
C06731=1029.068,353.183,-136.244,172.045,46.893,159.219
C06732=1029.077,353.430,-136.283,172.052,46.894,159.220
C06733=1029.084,353.676,-136.321,172.059,46.895,159.221
C06734=1029.092,353.924,-136.359,172.065,46.896,159.222
C06735=1029.100,354.170,-136.397,172.072,46.897,159.223
C06736=1029.108,354.418,-136.435,172.079,46.898,159.224
C06737=1029.116,354.665,-136.473,172.085,46.899,159.225
C06738=1029.124,354.912,-136.512,172.091,46.900,159.227
C06739=1029.132,355.158,-136.549,172.099,46.901,159.228
C06740=1029.140,355.405,-136.588,172.105,46.903,159.229
C06741=1029.148,355.652,-136.626,172.113,46.903,159.230
C06742=1029.156,355.900,-136.664,172.119,46.904,159.231
C06743=1029.163,356.146,-136.702,172.125,46.906,159.232
C06744=1029.171,356.393,-136.741,172.133,46.907,159.233
C06745=1029.180,356.641,-136.779,172.139,46.908,159.234
C06746=1029.187,356.887,-136.818,172.146,46.909,159.236
C06747=1029.195,357.134,-136.856,172.153,46.910,159.237
C06748=1029.203,357.381,-136.894,172.160,46.912,159.238
C06749=1029.211,357.628,-136.933,172.166,46.913,159.239
C06750=1029.219,357.875,-136.972,172.174,46.914,159.240
C06751=1029.227,358.121,-137.011,172.180,46.915,159.241
C06752=1029.235,358.368,-137.049,172.188,46.917,159.243
C06753=1029.243,358.616,-137.088,172.194,46.918,159.244
C06754=1029.251,358.862,-137.126,172.201,46.919,159.245
C06755=1029.259,359.109,-137.165,172.208,46.920,159.246
C06756=1029.267,359.356,-137.204,172.214,46.922,159.247
C06757=1029.276,359.603,-137.243,172.222,46.923,159.248
C06758=1029.283,359.850,-137.281,172.229,46.924,159.250
C06759=1029.292,360.096,-137.320,172.236,46.926,159.251
C06760=1029.300,360.344,-137.359,172.243,46.926,159.252
C06761=1029.308,360.591,-137.397,172.250,46.928,159.253
C06762=1029.316,360.837,-137.436,172.257,46.929,159.254
C06763=1029.324,361.084,-137.475,172.264,46.931,159.256
C06764=1029.332,361.331,-137.515,172.271,46.932,159.257
C06765=1029.340,361.578,-137.554,172.278,46.933,159.258
C06766=1029.348,361.825,-137.593,172.285,46.935,159.259
C06767=1029.356,362.071,-137.632,172.292,46.937,159.261
C06768=1029.363,362.318,-137.671,172.299,46.938,159.262
C06769=1029.372,362.565,-137.710,172.307,46.939,159.263
C06770=1029.380,362.811,-137.750,172.313,46.941,159.264
C06771=1029.389,363.058,-137.788,172.321,46.942,159.266
C06772=1029.396,363.305,-137.828,172.328,46.944,159.267
C06773=1029.405,363.552,-137.868,172.335,46.945,159.268
C06774=1029.413,363.798,-137.906,172.343,46.947,159.269
C06775=1029.420,364.045,-137.946,172.349,46.948,159.271
C06776=1029.428,364.292,-137.985,172.357,46.950,159.272
C06777=1029.438,364.577,-138.031,172.365,46.952,159.273
C06778=1029.447,364.861,-138.076,172.374,46.953,159.275
C06779=1029.457,365.146,-138.122,172.382,46.955,159.276
C06780=1029.466,365.430,-138.168,172.390,46.957,159.278
C06781=1029.475,365.677,-138.207,172.398,46.958,159.279
C06782=1029.483,365.924,-138.246,172.405,46.960,159.280
C06783=1029.491,366.170,-138.286,172.412,46.962,159.282
C06784=1029.500,366.417,-138.326,172.420,46.963,159.283
C06785=1029.508,366.664,-138.365,172.427,46.965,159.284
C06786=1029.516,366.910,-138.404,172.434,46.966,159.286
C06787=1029.525,367.158,-138.444,172.442,46.968,159.287
C06788=1029.533,367.404,-138.484,172.450,46.970,159.289
C06789=1029.542,367.651,-138.523,172.456,46.972,159.290
C06790=1029.550,367.897,-138.564,172.464,46.973,159.291
C06791=1029.558,368.144,-138.603,172.472,46.975,159.293
C06792=1029.567,368.391,-138.642,172.479,46.976,159.294
C06793=1029.575,368.638,-138.683,172.486,46.978,159.295
C06794=1029.584,368.884,-138.723,172.494,46.980,159.297
C06795=1029.592,369.131,-138.762,172.501,46.981,159.298
C06796=1029.600,369.378,-138.802,172.509,46.983,159.299
C06797=1029.614,369.770,-138.866,172.521,46.986,159.302
C06798=1029.627,370.162,-138.931,172.533,46.989,159.304
C06799=1029.640,370.555,-138.994,172.546,46.992,159.306
C06800=1029.653,370.947,-139.059,172.558,46.995,159.308
C06801=1029.662,371.193,-139.099,172.566,46.997,159.310
C06802=1029.670,371.441,-139.139,172.572,46.999,159.311
C06803=1029.678,371.687,-139.180,172.580,47.001,159.313
C06804=1029.687,371.933,-139.220,172.588,47.003,159.314
C06805=1029.695,372.180,-139.261,172.596,47.004,159.316
C06806=1029.704,372.427,-139.300,172.604,47.006,159.317
C06807=1029.712,372.673,-139.341,172.612,47.008,159.319
C06808=1029.721,372.920,-139.382,172.619,47.010,159.320
C06809=1029.729,373.166,-139.422,172.627,47.012,159.322
C06810=1029.738,373.413,-139.463,172.635,47.014,159.323
C06811=1029.746,373.659,-139.503,172.643,47.016,159.324
C06812=1029.755,373.906,-139.544,172.651,47.018,159.326
C06813=1029.763,374.152,-139.584,172.659,47.019,159.327
C06814=1029.771,374.398,-139.625,172.666,47.022,159.329
C06815=1029.781,374.645,-139.665,172.674,47.024,159.331
C06816=1029.789,374.892,-139.706,172.682,47.026,159.332
C06817=1029.797,375.138,-139.747,172.690,47.028,159.334
C06818=1029.807,375.385,-139.787,172.698,47.030,159.335
C06819=1029.815,375.631,-139.828,172.705,47.032,159.336
C06820=1029.823,375.878,-139.869,172.715,47.034,159.338
C06821=1029.832,376.124,-139.910,172.723,47.036,159.340
C06822=1029.841,376.371,-139.951,172.730,47.038,159.341
C06823=1029.850,376.618,-139.992,172.739,47.040,159.343
C06824=1029.859,376.863,-140.032,172.747,47.042,159.344
C06825=1029.867,377.110,-140.073,172.754,47.044,159.346
C06826=1029.876,377.357,-140.114,172.763,47.047,159.347
C06827=1029.885,377.602,-140.155,172.771,47.049,159.349
C06828=1029.894,377.849,-140.196,172.779,47.051,159.351
C06829=1029.903,378.096,-140.238,172.787,47.053,159.352
C06830=1029.911,378.342,-140.279,172.795,47.056,159.354
C06831=1029.920,378.588,-140.320,172.803,47.057,159.355
C06832=1029.929,378.835,-140.362,172.811,47.060,159.357
C06833=1029.936,379.060,-140.400,172.819,47.062,159.358
C06834=1029.944,379.287,-140.437,172.827,47.064,159.360
C06835=1029.952,379.512,-140.475,172.834,47.067,159.362
C06836=1029.960,379.738,-140.513,172.842,47.068,159.363
C06837=1029.968,379.964,-140.551,172.850,47.070,159.365
C06838=1029.976,380.189,-140.589,172.857,47.072,159.366
C06839=1029.984,380.416,-140.628,172.864,47.074,159.367
C06840=1029.992,380.641,-140.665,172.873,47.077,159.369
C06841=1030.001,380.887,-140.707,172.881,47.079,159.371
C06842=1030.010,381.134,-140.749,172.889,47.081,159.372
C06843=1030.019,381.380,-140.791,172.897,47.084,159.374
C06844=1030.028,381.627,-140.832,172.905,47.086,159.376
C06845=1030.037,381.873,-140.874,172.914,47.088,159.377
C06846=1030.046,382.119,-140.916,172.923,47.091,159.379
C06847=1030.054,382.366,-140.957,172.931,47.093,159.381
C06848=1030.063,382.612,-140.999,172.939,47.096,159.382
C06849=1030.072,382.858,-141.041,172.948,47.098,159.384
C06850=1030.081,383.104,-141.084,172.956,47.100,159.386
C06851=1030.090,383.351,-141.126,172.965,47.104,159.388
C06852=1030.099,383.597,-141.167,172.974,47.106,159.389
C06853=1030.108,383.844,-141.209,172.982,47.108,159.391
C06854=1030.117,384.089,-141.251,172.991,47.111,159.393
C06855=1030.126,384.336,-141.293,173.000,47.113,159.395
C06856=1030.135,384.582,-141.335,173.008,47.116,159.396
C06857=1030.144,384.828,-141.377,173.017,47.118,159.398
C06858=1030.153,385.074,-141.419,173.026,47.120,159.400
C06859=1030.162,385.320,-141.461,173.034,47.124,159.402
C06860=1030.172,385.567,-141.504,173.044,47.126,159.403
C06861=1030.181,385.813,-141.545,173.052,47.128,159.405
C06862=1030.190,386.059,-141.588,173.061,47.131,159.407
C06863=1030.199,386.305,-141.629,173.070,47.133,159.409
C06864=1030.208,386.551,-141.672,173.078,47.136,159.411
C06865=1030.218,386.798,-141.715,173.087,47.139,159.412
C06866=1030.227,387.044,-141.756,173.096,47.142,159.414
C06867=1030.236,387.290,-141.799,173.105,47.144,159.416
C06868=1030.245,387.536,-141.842,173.114,47.147,159.418
C06869=1030.254,387.782,-141.885,173.123,47.150,159.420
C06870=1030.264,388.028,-141.927,173.132,47.153,159.422
C06871=1030.272,388.275,-141.969,173.141,47.155,159.424
C06872=1030.282,388.521,-142.012,173.149,47.158,159.425
C06873=1030.291,388.767,-142.055,173.159,47.160,159.427
C06874=1030.300,389.013,-142.097,173.167,47.164,159.429
C06875=1030.309,389.259,-142.140,173.177,47.166,159.431
C06876=1030.319,389.505,-142.183,173.187,47.169,159.433
C06877=1030.328,389.751,-142.226,173.195,47.172,159.435
C06878=1030.337,389.997,-142.269,173.205,47.175,159.437
C06879=1030.346,390.243,-142.312,173.213,47.178,159.439
C06880=1030.356,390.489,-142.355,173.223,47.180,159.441
C06881=1030.365,390.735,-142.398,173.232,47.183,159.443
C06882=1030.375,390.981,-142.441,173.241,47.186,159.444
C06883=1030.383,391.227,-142.484,173.250,47.189,159.446
C06884=1030.393,391.473,-142.527,173.260,47.192,159.448
C06885=1030.402,391.719,-142.571,173.269,47.195,159.450
C06886=1030.412,391.965,-142.614,173.278,47.198,159.452
C06887=1030.421,392.211,-142.657,173.288,47.201,159.454
C06888=1030.431,392.457,-142.700,173.297,47.204,159.456
C06889=1030.440,392.703,-142.744,173.306,47.207,159.458
C06890=1030.449,392.949,-142.787,173.316,47.210,159.460
C06891=1030.459,393.195,-142.831,173.326,47.213,159.462
C06892=1030.468,393.442,-142.874,173.334,47.216,159.464
C06893=1030.478,393.684,-142.916,173.344,47.219,159.466
C06894=1030.487,393.928,-142.960,173.354,47.222,159.468
C06895=1030.496,394.172,-143.003,173.362,47.225,159.470
C06896=1030.506,394.415,-143.046,173.372,47.228,159.472
C06897=1030.515,394.658,-143.089,173.382,47.231,159.475
C06898=1030.524,394.902,-143.133,173.391,47.234,159.476
C06899=1030.534,395.146,-143.175,173.400,47.238,159.479
C06900=1030.544,395.389,-143.219,173.410,47.241,159.481
C06901=1030.553,395.636,-143.263,173.420,47.244,159.483
C06902=1030.563,395.881,-143.307,173.430,47.247,159.485
C06903=1030.572,396.128,-143.351,173.439,47.250,159.487
C06904=1030.581,396.373,-143.394,173.449,47.253,159.489
C06905=1030.592,396.618,-143.439,173.459,47.257,159.491
C06906=1030.601,396.864,-143.483,173.469,47.260,159.493
C06907=1030.611,397.110,-143.527,173.479,47.263,159.495
C06908=1030.621,397.356,-143.570,173.489,47.266,159.498
C06909=1030.630,397.602,-143.615,173.499,47.270,159.500
C06910=1030.640,397.848,-143.659,173.509,47.273,159.502
C06911=1030.650,398.094,-143.703,173.519,47.276,159.504
C06912=1030.659,398.340,-143.747,173.528,47.279,159.506
C06913=1030.669,398.585,-143.792,173.538,47.283,159.508
C06914=1030.679,398.831,-143.835,173.548,47.287,159.511
C06915=1030.689,399.077,-143.880,173.558,47.290,159.513
C06916=1030.698,399.323,-143.924,173.568,47.293,159.515
C06917=1030.708,399.568,-143.969,173.578,47.297,159.517
C06918=1030.718,399.814,-144.013,173.588,47.300,159.519
C06919=1030.729,400.060,-144.058,173.598,47.303,159.522
C06920=1030.738,400.306,-144.103,173.608,47.307,159.524
C06921=1030.748,400.551,-144.147,173.618,47.310,159.526
C06922=1030.757,400.798,-144.192,173.629,47.314,159.528
C06923=1030.767,401.043,-144.236,173.640,47.318,159.531
C06924=1030.777,401.289,-144.281,173.650,47.321,159.533
C06925=1030.788,401.535,-144.326,173.660,47.325,159.535
C06926=1030.798,401.780,-144.371,173.670,47.328,159.538
C06927=1030.807,402.026,-144.415,173.680,47.332,159.540
C06928=1030.818,402.272,-144.461,173.691,47.335,159.542
C06929=1030.827,402.517,-144.505,173.701,47.339,159.545
C06930=1030.837,402.763,-144.550,173.712,47.343,159.547
C06931=1030.847,403.009,-144.595,173.722,47.347,159.549
C06932=1030.856,403.255,-144.641,173.733,47.350,159.552
C06933=1030.866,403.500,-144.686,173.743,47.354,159.554
C06934=1030.877,403.746,-144.732,173.753,47.358,159.556
C06935=1030.886,403.991,-144.776,173.764,47.361,159.559
C06936=1030.897,404.237,-144.822,173.775,47.365,159.561
C06937=1030.907,404.483,-144.867,173.785,47.369,159.564
C06938=1030.917,404.729,-144.912,173.796,47.372,159.566
C06939=1030.927,404.974,-144.958,173.807,47.376,159.568
C06940=1030.937,405.220,-145.003,173.817,47.380,159.571
C06941=1030.947,405.465,-145.049,173.828,47.384,159.573
C06942=1030.958,405.711,-145.094,173.839,47.387,159.576
C06943=1030.968,405.956,-145.139,173.850,47.391,159.578
C06944=1030.978,406.202,-145.186,173.860,47.395,159.581
C06945=1030.988,406.448,-145.231,173.872,47.399,159.583
C06946=1030.998,406.693,-145.277,173.882,47.403,159.586
C06947=1031.009,406.938,-145.322,173.894,47.407,159.588
C06948=1031.019,407.184,-145.368,173.904,47.411,159.591
C06949=1031.030,407.430,-145.414,173.915,47.415,159.593
C06950=1031.040,407.675,-145.459,173.926,47.419,159.596
C06951=1031.050,407.921,-145.505,173.937,47.422,159.598
C06952=1031.061,408.166,-145.551,173.948,47.427,159.601
C06953=1031.072,408.428,-145.600,173.961,47.431,159.604
C06954=1031.083,408.691,-145.650,173.972,47.435,159.606
C06955=1031.094,408.953,-145.699,173.984,47.440,159.609
C06956=1031.106,409.216,-145.748,173.996,47.444,159.612
C06957=1031.116,409.462,-145.794,174.007,47.448,159.614
C06958=1031.126,409.707,-145.840,174.019,47.452,159.617
C06959=1031.137,409.953,-145.886,174.029,47.456,159.619
C06960=1031.148,410.198,-145.932,174.041,47.460,159.622
C06961=1031.159,410.443,-145.978,174.053,47.464,159.625
C06962=1031.169,410.689,-146.024,174.064,47.468,159.627
C06963=1031.179,410.934,-146.071,174.075,47.473,159.630
C06964=1031.190,411.180,-146.117,174.087,47.477,159.633
C06965=1031.200,411.425,-146.165,174.099,47.481,159.635
C06966=1031.211,411.670,-146.211,174.110,47.485,159.638
C06967=1031.222,411.916,-146.257,174.122,47.490,159.641
C06968=1031.232,412.161,-146.304,174.133,47.494,159.643
C06969=1031.243,412.407,-146.351,174.144,47.498,159.646
C06970=1031.253,412.653,-146.398,174.156,47.502,159.649
C06971=1031.264,412.898,-146.444,174.168,47.507,159.652
C06972=1031.274,413.143,-146.492,174.180,47.511,159.654
C06973=1031.285,413.388,-146.538,174.191,47.515,159.657
C06974=1031.296,413.634,-146.586,174.203,47.520,159.660
C06975=1031.307,413.879,-146.632,174.215,47.524,159.663
C06976=1031.318,414.124,-146.679,174.227,47.529,159.666
C06977=1031.329,414.370,-146.727,174.239,47.533,159.668
C06978=1031.340,414.615,-146.773,174.251,47.537,159.671
C06979=1031.351,414.861,-146.821,174.263,47.542,159.674
C06980=1031.361,415.106,-146.868,174.275,47.546,159.677
C06981=1031.372,415.350,-146.915,174.287,47.550,159.680
C06982=1031.384,415.596,-146.962,174.299,47.555,159.683
C06983=1031.394,415.841,-147.010,174.312,47.560,159.686
C06984=1031.406,416.086,-147.057,174.324,47.564,159.688
C06985=1031.417,416.332,-147.104,174.335,47.569,159.691
C06986=1031.427,416.577,-147.152,174.347,47.573,159.694
C06987=1031.438,416.823,-147.200,174.361,47.578,159.697
C06988=1031.449,417.068,-147.246,174.373,47.583,159.700
C06989=1031.460,417.313,-147.295,174.385,47.588,159.703
C06990=1031.471,417.558,-147.343,174.397,47.592,159.706
C06991=1031.483,417.803,-147.390,174.410,47.597,159.709
C06992=1031.494,418.049,-147.438,174.422,47.601,159.712
C06993=1031.505,418.294,-147.486,174.434,47.606,159.715
C06994=1031.515,418.539,-147.534,174.447,47.611,159.718
C06995=1031.527,418.784,-147.582,174.460,47.616,159.721
C06996=1031.538,419.029,-147.630,174.473,47.621,159.724
C06997=1031.549,419.275,-147.679,174.485,47.625,159.727
C06998=1031.561,419.520,-147.726,174.497,47.630,159.730
C06999=1031.571,419.764,-147.774,174.510,47.635,159.733
C07000=1031.583,420.010,-147.822,174.523,47.640,159.736
C07001=1031.594,420.255,-147.871,174.536,47.644,159.739
C07002=1031.606,420.499,-147.919,174.550,47.650,159.743
C07003=1031.617,420.745,-147.967,174.562,47.655,159.746
C07004=1031.628,420.990,-148.016,174.575,47.659,159.749
C07005=1031.640,421.235,-148.064,174.587,47.664,159.752
C07006=1031.651,421.480,-148.112,174.601,47.669,159.755
C07007=1031.663,421.725,-148.161,174.614,47.674,159.758
C07008=1031.674,421.970,-148.210,174.627,47.679,159.761
C07009=1031.686,422.215,-148.257,174.640,47.684,159.765
C07010=1031.698,422.461,-148.307,174.654,47.689,159.768
C07011=1031.709,422.705,-148.356,174.666,47.694,159.771
C07012=1031.720,422.951,-148.404,174.680,47.699,159.774
C07013=1031.733,423.223,-148.459,174.695,47.705,159.778
C07014=1031.746,423.496,-148.514,174.710,47.710,159.781
C07015=1031.759,423.768,-148.568,174.725,47.716,159.785
C07016=1031.772,424.041,-148.623,174.740,47.722,159.789
C07017=1031.784,424.286,-148.672,174.753,47.727,159.792
C07018=1031.795,424.531,-148.721,174.766,47.732,159.795
C07019=1031.807,424.776,-148.770,174.780,47.738,159.799
C07020=1031.819,425.021,-148.819,174.794,47.743,159.802
C07021=1031.830,425.266,-148.868,174.808,47.748,159.805
C07022=1031.841,425.511,-148.917,174.821,47.754,159.809
C07023=1031.854,425.756,-148.968,174.835,47.759,159.812
C07024=1031.865,426.000,-149.017,174.848,47.764,159.815
C07025=1031.878,426.245,-149.066,174.862,47.770,159.819
C07026=1031.890,426.490,-149.115,174.877,47.774,159.822
C07027=1031.902,426.735,-149.164,174.891,47.780,159.826
C07028=1031.913,426.979,-149.214,174.905,47.785,159.829
C07029=1031.926,427.224,-149.264,174.919,47.791,159.833
C07030=1031.937,427.470,-149.314,174.933,47.796,159.836
C07031=1031.949,427.714,-149.364,174.947,47.802,159.840
C07032=1031.961,427.959,-149.414,174.962,47.807,159.843
C07033=1031.973,428.203,-149.464,174.975,47.813,159.847
C07034=1031.985,428.448,-149.514,174.989,47.818,159.850
C07035=1031.996,428.693,-149.565,175.004,47.824,159.854
C07036=1032.009,428.938,-149.615,175.019,47.830,159.858
C07037=1032.020,429.182,-149.664,175.033,47.835,159.861
C07038=1032.033,429.427,-149.714,175.048,47.841,159.865
C07039=1032.045,429.671,-149.765,175.062,47.846,159.868
C07040=1032.057,429.916,-149.816,175.077,47.852,159.872
C07041=1032.069,430.161,-149.866,175.091,47.858,159.876
C07042=1032.082,430.406,-149.916,175.106,47.863,159.879
C07043=1032.094,430.650,-149.967,175.120,47.869,159.883
C07044=1032.107,430.895,-150.017,175.135,47.874,159.887
C07045=1032.118,431.139,-150.068,175.150,47.881,159.890
C07046=1032.131,431.384,-150.119,175.165,47.886,159.894
C07047=1032.143,431.628,-150.169,175.180,47.892,159.898
C07048=1032.156,431.873,-150.219,175.194,47.898,159.902
C07049=1032.168,432.117,-150.270,175.210,47.904,159.905
C07050=1032.181,432.361,-150.321,175.225,47.909,159.909
C07051=1032.193,432.606,-150.372,175.241,47.915,159.913
C07052=1032.205,432.850,-150.423,175.255,47.921,159.917
C07053=1032.218,433.096,-150.474,175.270,47.927,159.921
C07054=1032.231,433.340,-150.525,175.286,47.933,159.924
C07055=1032.244,433.584,-150.575,175.301,47.939,159.928
C07056=1032.256,433.827,-150.627,175.317,47.945,159.932
C07057=1032.269,434.073,-150.679,175.332,47.951,159.936
C07058=1032.282,434.317,-150.729,175.348,47.957,159.940
C07059=1032.294,434.562,-150.781,175.363,47.963,159.944
C07060=1032.307,434.806,-150.833,175.379,47.969,159.948
C07061=1032.320,435.050,-150.884,175.394,47.975,159.952
C07062=1032.332,435.295,-150.935,175.410,47.981,159.956
C07063=1032.345,435.539,-150.987,175.426,47.987,159.960
C07064=1032.358,435.783,-151.039,175.441,47.994,159.964
C07065=1032.370,436.027,-151.090,175.458,47.999,159.968
C07066=1032.384,436.272,-151.142,175.474,48.006,159.972
C07067=1032.397,436.516,-151.195,175.490,48.012,159.976
C07068=1032.410,436.760,-151.246,175.505,48.018,159.980
C07069=1032.422,437.005,-151.298,175.522,48.024,159.984
C07070=1032.436,437.249,-151.350,175.538,48.030,159.988
C07071=1032.448,437.493,-151.402,175.554,48.037,159.993
C07072=1032.462,437.737,-151.455,175.571,48.043,159.997
C07073=1032.475,437.996,-151.510,175.588,48.050,160.001
C07074=1032.489,438.256,-151.565,175.606,48.057,160.006
C07075=1032.503,438.516,-151.621,175.623,48.063,160.010
C07076=1032.517,438.774,-151.677,175.640,48.070,160.015
C07077=1032.530,439.019,-151.729,175.657,48.077,160.019
C07078=1032.544,439.263,-151.782,175.673,48.083,160.023
C07079=1032.557,439.507,-151.834,175.690,48.090,160.028
C07080=1032.570,439.751,-151.887,175.708,48.096,160.032
C07081=1032.584,439.995,-151.939,175.725,48.103,160.036
C07082=1032.597,440.239,-151.992,175.741,48.109,160.040
C07083=1032.610,440.483,-152.045,175.758,48.116,160.045
C07084=1032.624,440.727,-152.098,175.775,48.123,160.049
C07085=1032.637,440.971,-152.151,175.792,48.129,160.054
C07086=1032.651,441.214,-152.204,175.810,48.135,160.058
C07087=1032.664,441.458,-152.257,175.826,48.142,160.062
C07088=1032.677,441.703,-152.310,175.844,48.149,160.067
C07089=1032.691,441.947,-152.363,175.861,48.156,160.071
C07090=1032.704,442.191,-152.416,175.878,48.162,160.076
C07091=1032.718,442.434,-152.469,175.897,48.169,160.080
C07092=1032.732,442.678,-152.523,175.914,48.176,160.085
C07093=1032.745,442.922,-152.576,175.932,48.183,160.090
C07094=1032.759,443.165,-152.630,175.949,48.189,160.094
C07095=1032.773,443.409,-152.682,175.967,48.196,160.099
C07096=1032.787,443.653,-152.737,175.984,48.203,160.103
C07097=1032.802,443.895,-152.789,176.002,48.209,160.108
C07098=1032.817,444.139,-152.841,176.020,48.216,160.112
C07099=1032.832,444.382,-152.893,176.038,48.223,160.117
C07100=1032.849,444.627,-152.945,176.056,48.229,160.122
C07101=1032.865,444.869,-152.996,176.074,48.236,160.126
C07102=1032.881,445.113,-153.047,176.093,48.242,160.131
C07103=1032.899,445.357,-153.097,176.111,48.248,160.135
C07104=1032.917,445.602,-153.147,176.130,48.254,160.140
C07105=1032.935,445.845,-153.196,176.148,48.260,160.144
C07106=1032.954,446.089,-153.245,176.167,48.266,160.149
C07107=1032.974,446.333,-153.295,176.185,48.272,160.153
C07108=1032.994,446.577,-153.342,176.205,48.278,160.158
C07109=1033.015,446.822,-153.390,176.223,48.284,160.162
C07110=1033.036,447.066,-153.438,176.242,48.289,160.167
C07111=1033.057,447.310,-153.484,176.261,48.295,160.171
C07112=1033.079,447.555,-153.531,176.280,48.301,160.176
C07113=1033.102,447.800,-153.577,176.299,48.306,160.180
C07114=1033.125,448.044,-153.623,176.319,48.312,160.184
C07115=1033.149,448.289,-153.669,176.338,48.317,160.189
C07116=1033.173,448.534,-153.713,176.358,48.322,160.193
C07117=1033.197,448.779,-153.758,176.377,48.327,160.198
C07118=1033.222,449.024,-153.802,176.397,48.332,160.202
C07119=1033.248,449.268,-153.845,176.417,48.337,160.206
C07120=1033.274,449.514,-153.888,176.436,48.342,160.211
C07121=1033.300,449.759,-153.931,176.456,48.347,160.215
C07122=1033.328,450.004,-153.974,176.475,48.352,160.220
C07123=1033.355,450.250,-154.015,176.496,48.357,160.224
C07124=1033.383,450.494,-154.057,176.517,48.361,160.229
C07125=1033.412,450.740,-154.098,176.536,48.366,160.233
C07126=1033.441,450.986,-154.139,176.556,48.370,160.237
C07127=1033.471,451.231,-154.179,176.577,48.374,160.241
C07128=1033.501,451.476,-154.219,176.598,48.379,160.246
C07129=1033.532,451.722,-154.258,176.618,48.383,160.250
C07130=1033.563,451.968,-154.297,176.638,48.387,160.254
C07131=1033.595,452.214,-154.335,176.659,48.391,160.259
C07132=1033.627,452.458,-154.373,176.680,48.396,160.263
C07133=1033.667,452.758,-154.419,176.706,48.401,160.268
C07134=1033.707,453.056,-154.463,176.732,48.405,160.274
C07135=1033.423,453.120,-154.793,176.734,48.472,160.295
C07136=1033.386,452.845,-154.752,176.711,48.468,160.290
C07137=1033.349,452.570,-154.709,176.687,48.463,160.285
C07138=1033.316,452.324,-154.672,176.667,48.459,160.281
C07139=1033.284,452.079,-154.634,176.646,48.455,160.276
C07140=1033.252,451.833,-154.595,176.625,48.451,160.272
C07141=1033.222,451.586,-154.556,176.604,48.447,160.268
C07142=1033.191,451.342,-154.517,176.584,48.443,160.264
C07143=1033.161,451.097,-154.477,176.563,48.438,160.259
C07144=1033.132,450.851,-154.436,176.543,48.434,160.255
C07145=1033.103,450.606,-154.396,176.522,48.429,160.250
C07146=1033.074,450.360,-154.354,176.502,48.425,160.246
C07147=1033.047,450.116,-154.312,176.482,48.421,160.242
C07148=1033.019,449.870,-154.271,176.462,48.416,160.237
C07149=1032.992,449.625,-154.228,176.442,48.411,160.233
C07150=1032.966,449.380,-154.185,176.422,48.406,160.229
C07151=1032.940,449.134,-154.142,176.402,48.401,160.224
C07152=1032.914,448.889,-154.098,176.382,48.396,160.220
C07153=1032.890,448.644,-154.054,176.364,48.392,160.216
C07154=1032.865,448.400,-154.009,176.343,48.387,160.211
C07155=1032.841,448.155,-153.964,176.324,48.381,160.207
C07156=1032.818,447.910,-153.919,176.304,48.376,160.202
C07157=1032.795,447.666,-153.872,176.285,48.371,160.198
C07158=1032.773,447.421,-153.827,176.266,48.365,160.193
C07159=1032.750,447.176,-153.780,176.247,48.360,160.189
C07160=1032.730,446.932,-153.732,176.228,48.355,160.184
C07161=1032.709,446.688,-153.685,176.210,48.349,160.180
C07162=1032.678,446.313,-153.611,176.180,48.340,160.173
C07163=1032.648,445.939,-153.537,176.151,48.331,160.166
C07164=1032.620,445.566,-153.462,176.123,48.322,160.159
C07165=1032.592,445.193,-153.385,176.095,48.313,160.152
C07166=1032.574,444.949,-153.334,176.077,48.306,160.148
C07167=1032.558,444.706,-153.283,176.058,48.300,160.143
C07168=1032.542,444.462,-153.231,176.040,48.294,160.139
C07169=1032.527,444.219,-153.180,176.021,48.288,160.134
C07170=1032.511,443.975,-153.128,176.004,48.281,160.130
